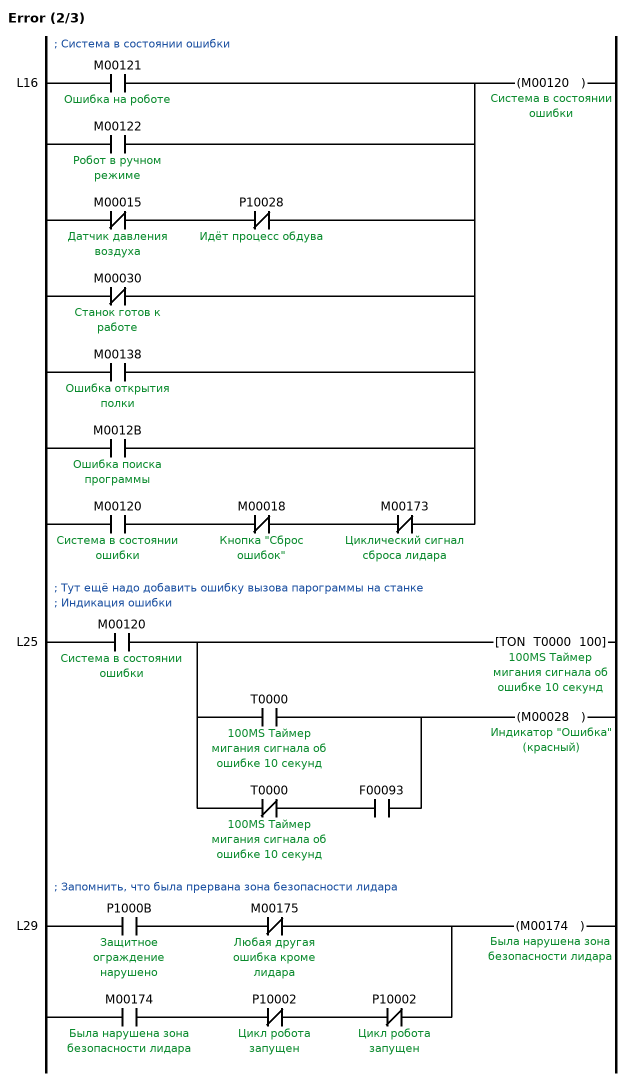
[picture p24: Error rungs L16-L29]
// Система в состоянии ошибки
; L16
LOAD      M00121	// Ошибка на роботе
OR        M00122	// Робот в ручном режиме
LOAD NOT  M00015	// Датчик давления воздуха
AND NOT   P10028	// Идёт процесс обдува
OR LOAD
OR NOT    M00030	// Станок готов к работе
OR        M00138	// Ошибка открытия полки
OR        M0012B	// Ошибка поиска программы
LOAD      M00120	// Система в состоянии ошибки
AND NOT   M00018	// Кнопка "Сброс ошибок"
AND NOT   M00173	// Циклический сигнал сброса лидара
OR LOAD
OUT       M00120	// Система в состоянии ошибки
// Тут ещё надо добавить ошибку вызова парограммы на станке
// Индикация ошибки
; L25
LOAD      M00120	// Система в состоянии ошибки
TON       T0000 100	// 100MS Таймер мигания сигнала об ошибке 10 секунд
LOAD      T0000	// 100MS Таймер мигания сигнала об ошибке 10 секунд
LOAD NOT  T0000	// 100MS Таймер мигания сигнала об ошибке 10 секунд
AND       F00093
OR LOAD
AND LOAD
OUT       M00028	// Индикатор "Ошибка" (красный)
// Запомнить, что была прервана зона безопасности лидара
; L29
LOAD      P1000B	// Защитное ограждение нарушено
AND NOT   M00175	// Любая другая ошибка кроме лидара
LOAD      M00174	// Была нарушена зона безопасности лидара
AND NOT   P10002	// Цикл робота запущен
AND NOT   P10002	// Цикл робота запущен
OR LOAD
OUT       M00174	// Была нарушена зона безопасности лидара

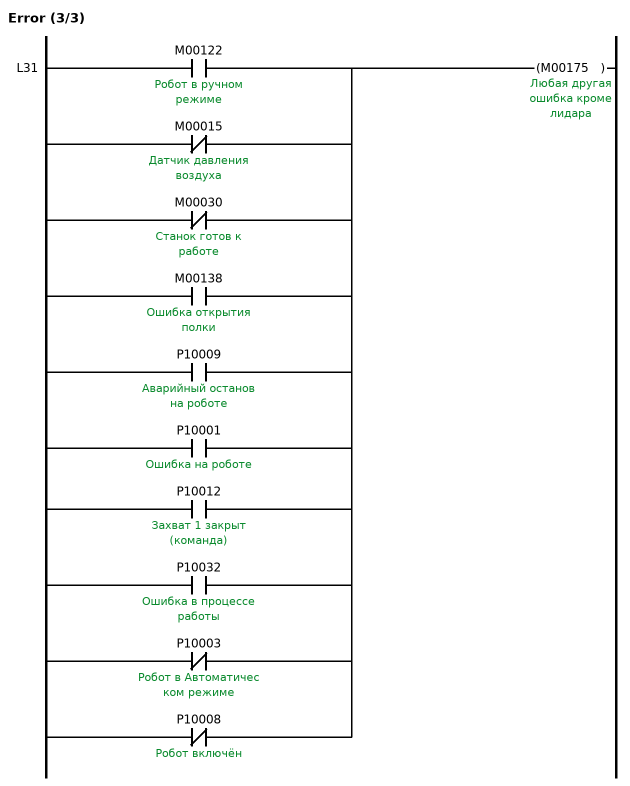
; L31
LOAD      M00122	// Робот в ручном режиме
OR NOT    M00015	// Датчик давления воздуха
OR NOT    M00030	// Станок готов к работе
OR        M00138	// Ошибка открытия полки
OR        P10009	// Аварийный останов на роботе
OR        P10001	// Ошибка на роботе
OR        P10012	// Захват 1 закрыт (команда)
OR        P10032	// Ошибка в процессе работы
OR NOT    P10003	// Робот в Автоматическом режиме
OR NOT    P10008	// Робот включён
OUT       M00175	// Любая другая ошибка кроме лидара

PROGRAM Shelves (task: Scan Program)

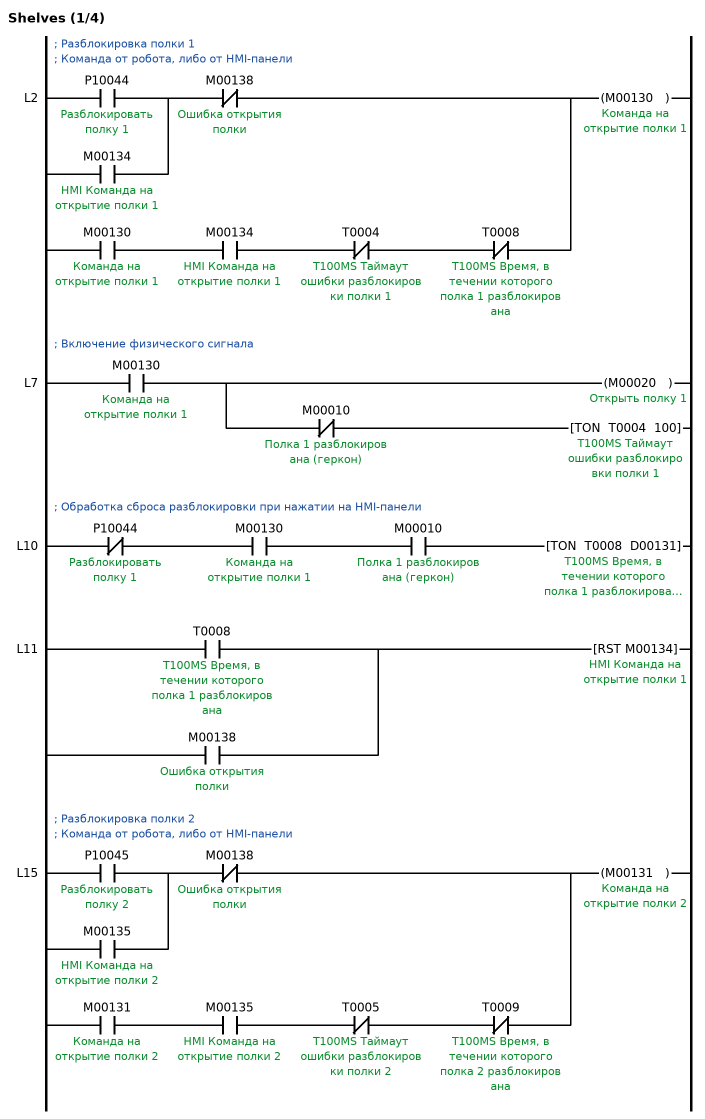
// Разблокировка полки 1
// Команда от робота, либо от HMI-панели
; L2
LOAD      P10044	// Разблокировать полку 1
OR        M00134	// HMI Команда на открытие полки 1
AND NOT   M00138	// Ошибка открытия полки
LOAD      M00130	// Команда на открытие полки 1
AND       M00134	// HMI Команда на открытие полки 1
AND NOT   T0004	// T100MS Таймаут ошибки разблокировки полки 1
AND NOT   T0008	// T100MS Время, в течении которого полка 1 разблокирована
OR LOAD
OUT       M00130	// Команда на открытие полки 1
// Включение физического сигнала
; L7
LOAD      M00130	// Команда на открытие полки 1
OUT       M00020	// Открыть полку 1
AND NOT   M00010	// Полка 1 разблокирована (геркон)
TON       T0004 100	// T100MS Таймаут ошибки разблокировки полки 1
// Обработка сброса разблокировки при нажатии на HMI-панели
; L10
LOAD NOT  P10044	// Разблокировать полку 1
AND       M00130	// Команда на открытие полки 1
AND       M00010	// Полка 1 разблокирована (геркон)
TON       T0008 D00131	// T100MS Время, в течении которого полка 1 разблокирована / HMI Время, в течении которого разблокирована полка после нажатия кнопки
; L11
LOAD      T0008	// T100MS Время, в течении которого полка 1 разблокирована
OR        M00138	// Ошибка открытия полки
RST       M00134	// HMI Команда на открытие полки 1
// Разблокировка полки 2
// Команда от робота, либо от HMI-панели
; L15
LOAD      P10045	// Разблокировать полку 2
OR        M00135	// HMI Команда на открытие полки 2
AND NOT   M00138	// Ошибка открытия полки
LOAD      M00131	// Команда на открытие полки 2
AND       M00135	// HMI Команда на открытие полки 2
AND NOT   T0005	// T100MS Таймаут ошибки разблокировки полки 2
AND NOT   T0009	// T100MS Время, в течении которого полка 2 разблокирована
OR LOAD
OUT       M00131	// Команда на открытие полки 2

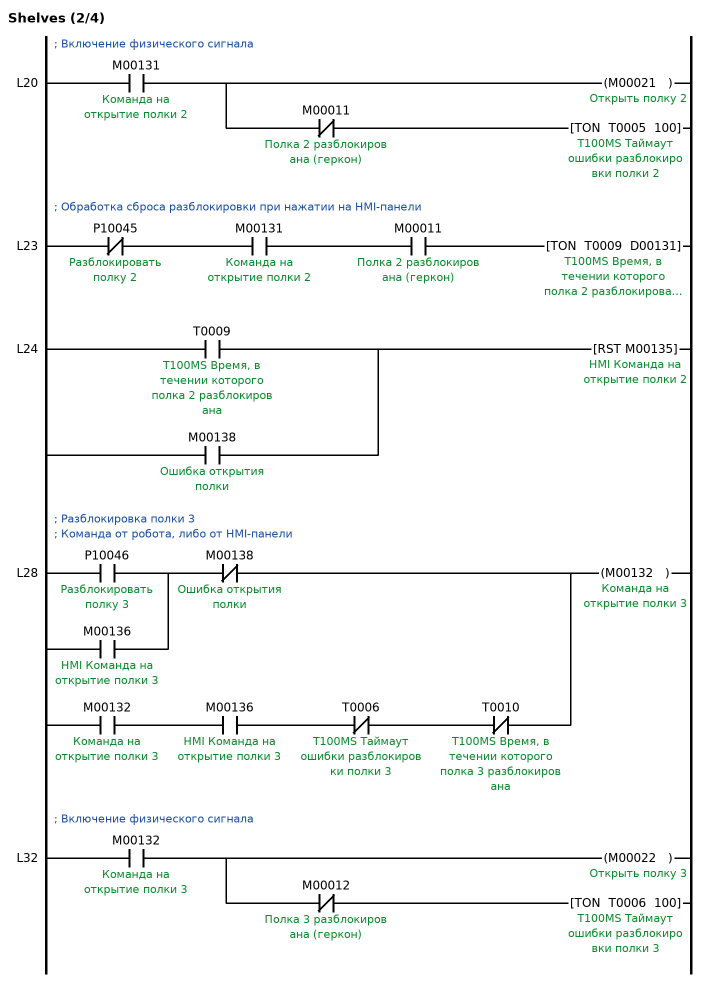
// Включение физического сигнала
; L20
LOAD      M00131	// Команда на открытие полки 2
OUT       M00021	// Открыть полку 2
AND NOT   M00011	// Полка 2 разблокирована (геркон)
TON       T0005 100	// T100MS Таймаут ошибки разблокировки полки 2
// Обработка сброса разблокировки при нажатии на HMI-панели
; L23
LOAD NOT  P10045	// Разблокировать полку 2
AND       M00131	// Команда на открытие полки 2
AND       M00011	// Полка 2 разблокирована (геркон)
TON       T0009 D00131	// T100MS Время, в течении которого полка 2 разблокирована / HMI Время, в течении которого разблокирована полка после нажатия кнопки
; L24
LOAD      T0009	// T100MS Время, в течении которого полка 2 разблокирована
OR        M00138	// Ошибка открытия полки
RST       M00135	// HMI Команда на открытие полки 2
// Разблокировка полки 3
// Команда от робота, либо от HMI-панели
; L28
LOAD      P10046	// Разблокировать полку 3
OR        M00136	// HMI Команда на открытие полки 3
AND NOT   M00138	// Ошибка открытия полки
LOAD      M00132	// Команда на открытие полки 3
AND       M00136	// HMI Команда на открытие полки 3
AND NOT   T0006	// T100MS Таймаут ошибки разблокировки полки 3
AND NOT   T0010	// T100MS Время, в течении которого полка 3 разблокирована
OR LOAD
OUT       M00132	// Команда на открытие полки 3
// Включение физического сигнала
; L32
LOAD      M00132	// Команда на открытие полки 3
OUT       M00022	// Открыть полку 3
AND NOT   M00012	// Полка 3 разблокирована (геркон)
TON       T0006 100	// T100MS Таймаут ошибки разблокировки полки 3

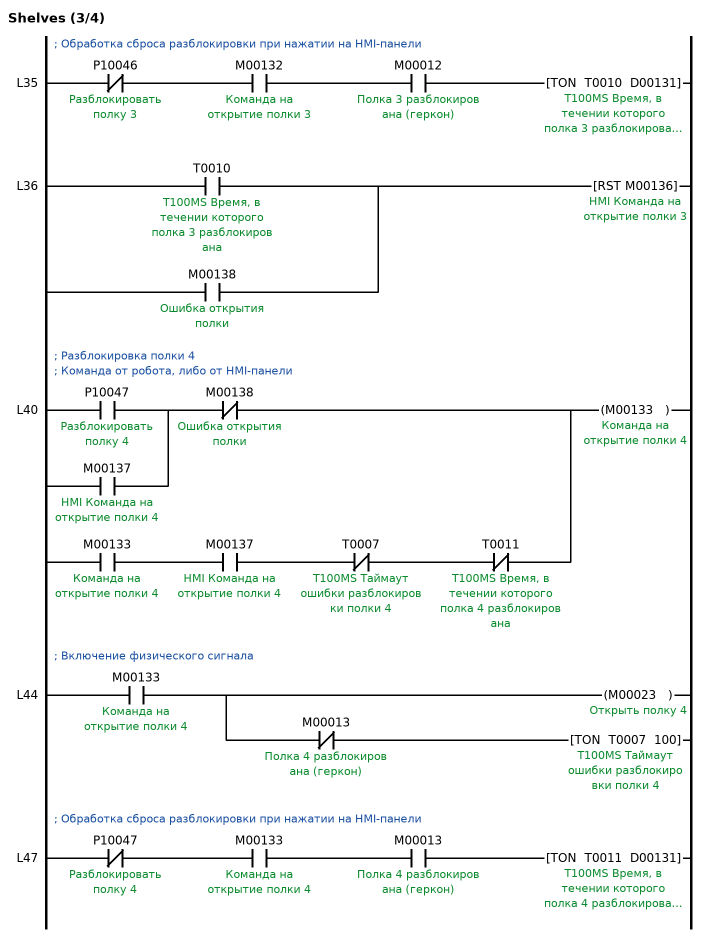
// Обработка сброса разблокировки при нажатии на HMI-панели
; L35
LOAD NOT  P10046	// Разблокировать полку 3
AND       M00132	// Команда на открытие полки 3
AND       M00012	// Полка 3 разблокирована (геркон)
TON       T0010 D00131	// T100MS Время, в течении которого полка 3 разблокирована / HMI Время, в течении которого разблокирована полка после нажатия кнопки
; L36
LOAD      T0010	// T100MS Время, в течении которого полка 3 разблокирована
OR        M00138	// Ошибка открытия полки
RST       M00136	// HMI Команда на открытие полки 3
// Разблокировка полки 4
// Команда от робота, либо от HMI-панели
; L40
LOAD      P10047	// Разблокировать полку 4
OR        M00137	// HMI Команда на открытие полки 4
AND NOT   M00138	// Ошибка открытия полки
LOAD      M00133	// Команда на открытие полки 4
AND       M00137	// HMI Команда на открытие полки 4
AND NOT   T0007	// T100MS Таймаут ошибки разблокировки полки 4
AND NOT   T0011	// T100MS Время, в течении которого полка 4 разблокирована
OR LOAD
OUT       M00133	// Команда на открытие полки 4
// Включение физического сигнала
; L44
LOAD      M00133	// Команда на открытие полки 4
OUT       M00023	// Открыть полку 4
AND NOT   M00013	// Полка 4 разблокирована (геркон)
TON       T0007 100	// T100MS Таймаут ошибки разблокировки полки 4
// Обработка сброса разблокировки при нажатии на HMI-панели
; L47
LOAD NOT  P10047	// Разблокировать полку 4
AND       M00133	// Команда на открытие полки 4
AND       M00013	// Полка 4 разблокирована (геркон)
TON       T0011 D00131	// T100MS Время, в течении которого полка 4 разблокирована / HMI Время, в течении которого разблокирована полка после нажатия кнопки

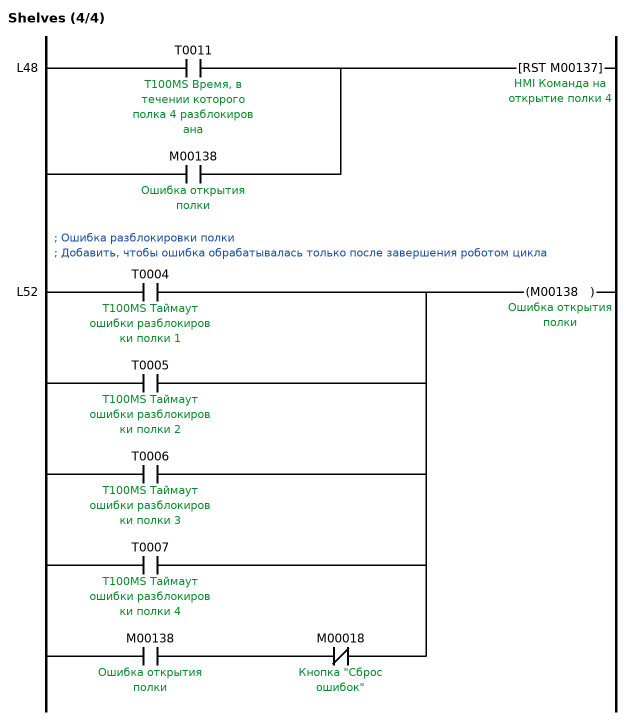
; L48
LOAD      T0011	// T100MS Время, в течении которого полка 4 разблокирована
OR        M00138	// Ошибка открытия полки
RST       M00137	// HMI Команда на открытие полки 4
// Ошибка разблокировки полки
// Добавить, чтобы ошибка обрабатывалась только после завершения роботом цикла
; L52
LOAD      T0004	// T100MS Таймаут ошибки разблокировки полки 1
OR        T0005	// T100MS Таймаут ошибки разблокировки полки 2
OR        T0006	// T100MS Таймаут ошибки разблокировки полки 3
OR        T0007	// T100MS Таймаут ошибки разблокировки полки 4
LOAD      M00138	// Ошибка открытия полки
AND NOT   M00018	// Кнопка "Сброс ошибок"
OR LOAD
OUT       M00138	// Ошибка открытия полки

PROGRAM Database (task: Scan Program)

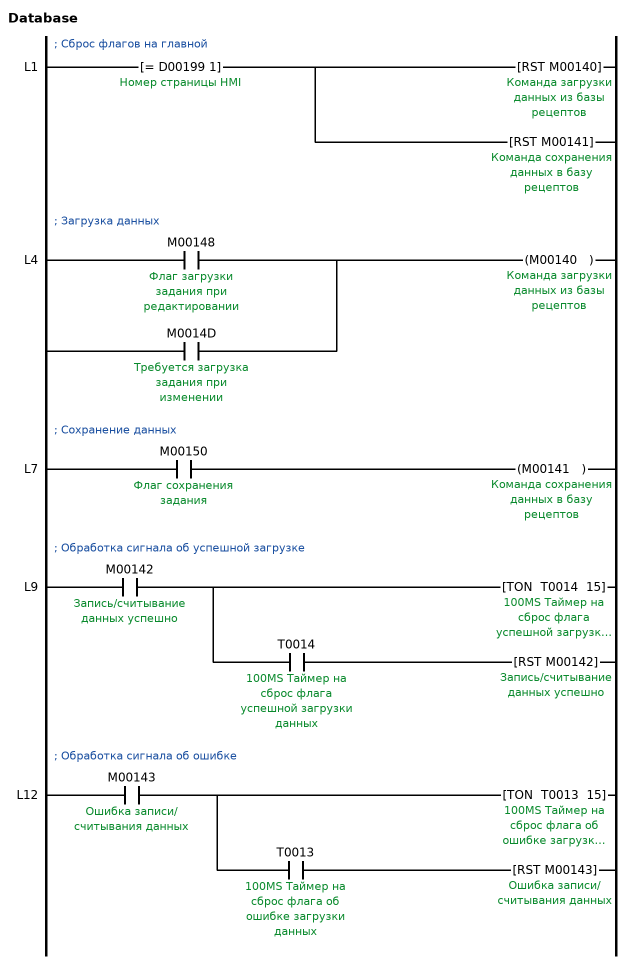
// Сброс флагов на главной
; L1
LOAD=     D00199 1	// Номер страницы HMI
RST       M00140	// Команда загрузки данных из базы рецептов
RST       M00141	// Команда сохранения данных в базу рецептов
// Загрузка данных
; L4
LOAD      M00148	// Флаг загрузки задания при редактировании
OR        M0014D	// Требуется загрузка задания при изменении
OUT       M00140	// Команда загрузки данных из базы рецептов
// Сохранение данных
; L7
LOAD      M00150	// Флаг сохранения задания
OUT       M00141	// Команда сохранения данных в базу рецептов
// Обработка сигнала об успешной загрузке
; L9
LOAD      M00142	// Запись/считывание данных успешно
TON       T0014 15	// 100MS Таймер на сброс флага успешной загрузки данных
AND       T0014	// 100MS Таймер на сброс флага успешной загрузки данных
RST       M00142	// Запись/считывание данных успешно
// Обработка сигнала об ошибке
; L12
LOAD      M00143	// Ошибка записи/считывания данных
TON       T0013 15	// 100MS Таймер на сброс флага об ошибке загрузки данных
AND       T0013	// 100MS Таймер на сброс флага об ошибке загрузки данных
RST       M00143	// Ошибка записи/считывания данных

PROGRAM HMI (task: Scan Program)

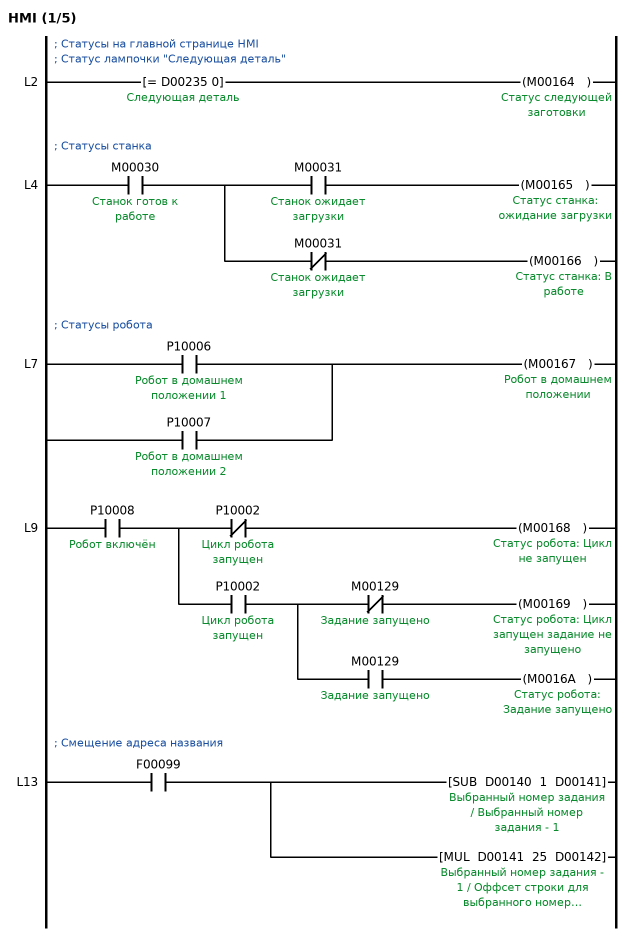
// Статусы на главной странице HMI
// Статус лампочки "Следующая деталь"
; L2
LOAD=     D00235 0	// Следующая деталь
OUT       M00164	// Статус следующей заготовки 
// Статусы станка
; L4
LOAD      M00030	// Станок готов к работе
MPUSH
AND       M00031	// Станок ожидает загрузки
OUT       M00165	// Статус станка: ожидание загрузки
MPOP
AND NOT   M00031	// Станок ожидает загрузки
OUT       M00166	// Статус станка: В работе
// Статусы робота
; L7
LOAD      P10006	// Робот в домашнем положении 1
OR        P10007	// Робот в домашнем положении 2
OUT       M00167	// Робот в домашнем положении
; L9
LOAD      P10008	// Робот включён
MPUSH
AND NOT   P10002	// Цикл робота запущен
OUT       M00168	// Статус робота: Цикл не запущен
MPOP
AND       P10002	// Цикл робота запущен
MPUSH
AND NOT   M00129	// Задание запущено
OUT       M00169	// Статус робота: Цикл запущен задание не запущено
MPOP
AND       M00129	// Задание запущено
OUT       M0016A	// Статус робота: Задание запущено
// Смещение адреса названия
; L13
LOAD      F00099
SUB       D00140 1 D00141	// Выбранный номер задания / Выбранный номер задания - 1
MUL       D00141 25 D00142	// Выбранный номер задания - 1 / Оффсет строки для выбранного номера названия

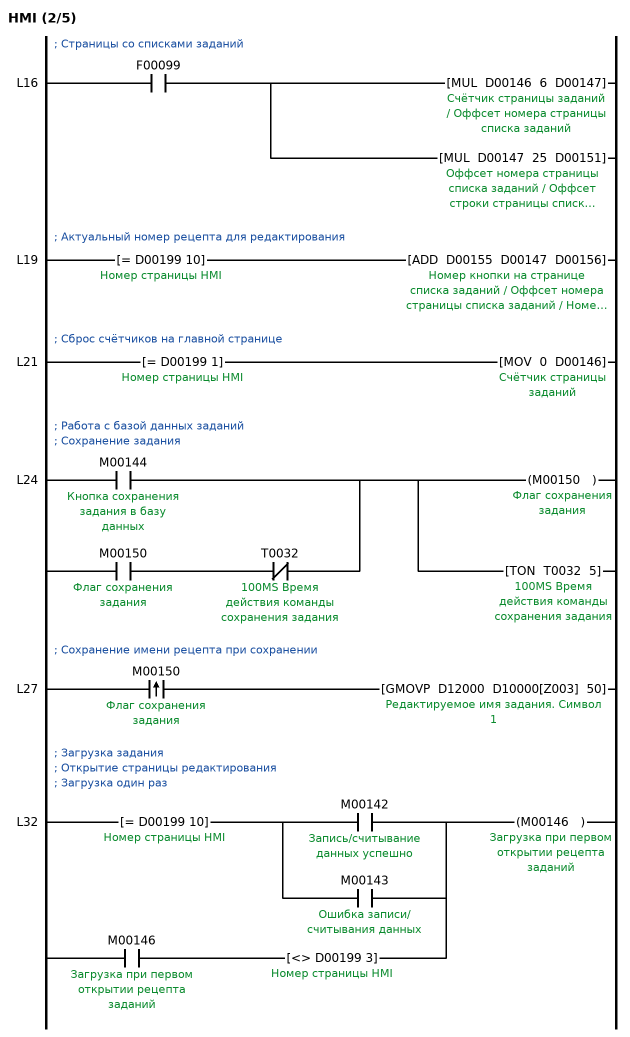
// Страницы со списками заданий
; L16
LOAD      F00099
MUL       D00146 6 D00147	// Счётчик страницы заданий / Оффсет номера страницы списка заданий
MUL       D00147 25 D00151	// Оффсет номера страницы списка заданий / Оффсет строки страницы списка заданий
// Актуальный номер рецепта для редактирования
; L19
LOAD=     D00199 10	// Номер страницы HMI
ADD       D00155 D00147 D00156	// Номер кнопки на странице списка заданий / Оффсет номера страницы списка заданий / Номер редактируемого задания
// Сброс счётчиков на главной странице
; L21
LOAD=     D00199 1	// Номер страницы HMI
MOV       0 D00146	// Счётчик страницы заданий
// Работа с базой данных заданий
// Сохранение задания
; L24
LOAD      M00144	// Кнопка сохранения задания в базу данных
LOAD      M00150	// Флаг сохранения задания
AND NOT   T0032	// 100MS Время действия команды сохранения задания
OR LOAD
OUT       M00150	// Флаг сохранения задания
TON       T0032 5	// 100MS Время действия команды сохранения задания
// Сохранение имени рецепта при сохранении
; L27
LOADP     M00150	// Флаг сохранения задания
GMOVP     D12000 D10000[Z003] 50	// Редактируемое имя задания. Символ 1
// Загрузка задания
// Открытие страницы редактирования
// Загрузка один раз
; L32
LOAD=     D00199 10	// Номер страницы HMI
LOAD      M00142	// Запись/считывание данных успешно
OR        M00143	// Ошибка записи/считывания данных
AND LOAD
LOAD      M00146	// Загрузка при первом открытии рецепта заданий
AND<>     D00199 3	// Номер страницы HMI
OR LOAD
OUT       M00146	// Загрузка при первом открытии рецепта заданий

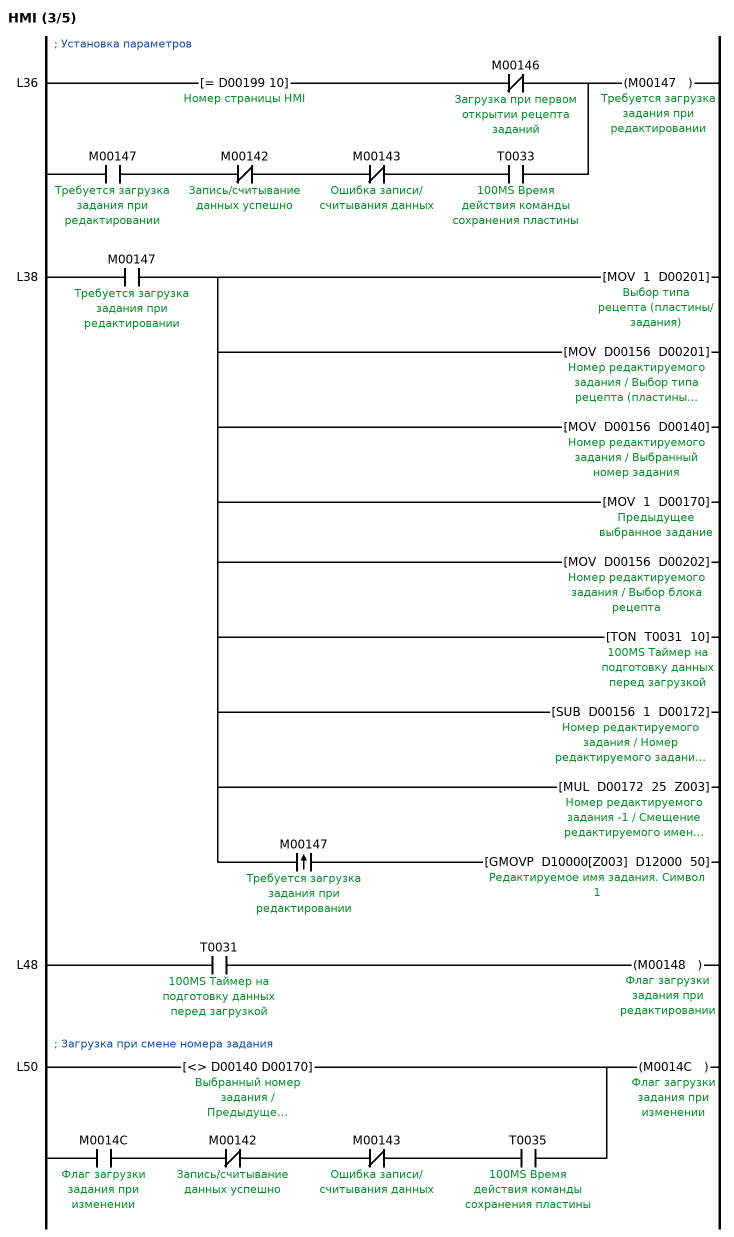
// Установка параметров
; L36
LOAD=     D00199 10	// Номер страницы HMI
AND NOT   M00146	// Загрузка при первом открытии рецепта заданий
LOAD      M00147	// Требуется загрузка задания при редактировании
AND NOT   M00142	// Запись/считывание данных успешно
AND NOT   M00143	// Ошибка записи/считывания данных
AND       T0033	// 100MS Время действия команды сохранения пластины
OR LOAD
OUT       M00147	// Требуется загрузка задания при редактировании
; L38
LOAD      M00147	// Требуется загрузка задания при редактировании
MOV       1 D00201	// Выбор типа рецепта (пластины/задания)
MOV       D00156 D00201	// Номер редактируемого задания / Выбор типа рецепта (пластины/задания)
MOV       D00156 D00140	// Номер редактируемого задания / Выбранный номер задания
MOV       1 D00170	// Предыдущее выбранное задание
MOV       D00156 D00202	// Номер редактируемого задания / Выбор блока рецепта
TON       T0031 10	// 100MS Таймер на подготовку данных перед загрузкой
SUB       D00156 1 D00172	// Номер редактируемого задания / Номер редактируемого задания -1
MUL       D00172 25 Z003	// Номер редактируемого задания -1 / Смещение редактируемого имени задания
ANDP      M00147	// Требуется загрузка задания при редактировании
GMOVP     D10000[Z003] D12000 50	// Редактируемое имя задания. Символ 1
; L48
LOAD      T0031	// 100MS Таймер на подготовку данных перед загрузкой
OUT       M00148	// Флаг загрузки задания при редактировании
// Загрузка при смене номера задания
; L50
LOAD<>    D00140 D00170	// Выбранный номер задания / Предыдущее выбранное задание
LOAD      M0014C	// Флаг загрузки задания при изменении
AND NOT   M00142	// Запись/считывание данных успешно
AND NOT   M00143	// Ошибка записи/считывания данных
AND       T0035	// 100MS Время действия команды сохранения пластины
OR LOAD
OUT       M0014C	// Флаг загрузки задания при изменении

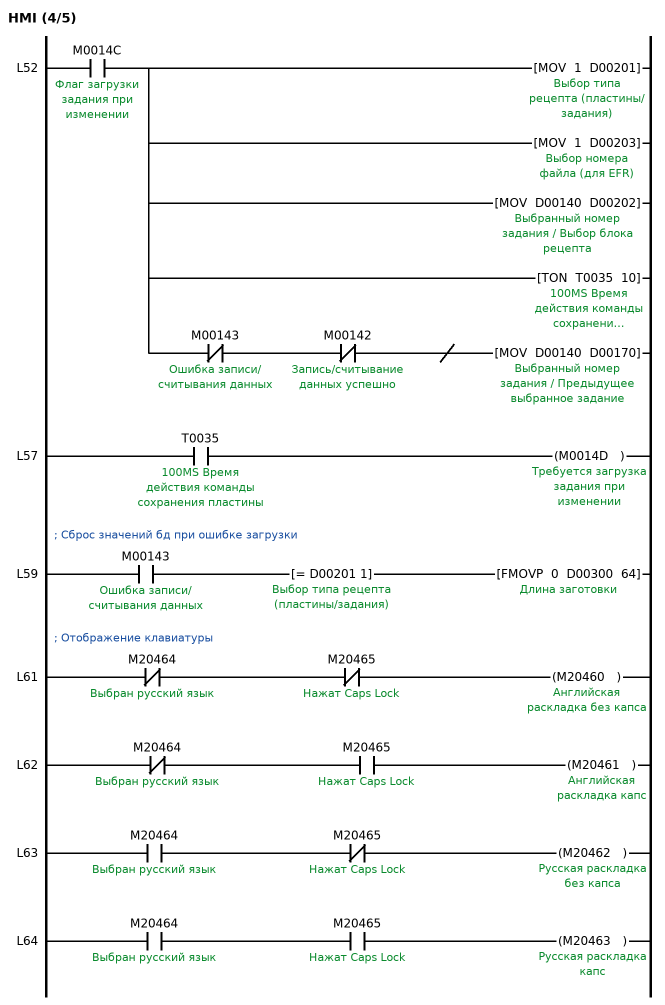
; L52
LOAD      M0014C	// Флаг загрузки задания при изменении
MOV       1 D00201	// Выбор типа рецепта (пластины/задания)
MOV       1 D00203	// Выбор номера файла (для EFR)
MOV       D00140 D00202	// Выбранный номер задания / Выбор блока рецепта
TON       T0035 10	// 100MS Время действия команды сохранения пластины
AND NOT   M00143	// Ошибка записи/считывания данных
AND NOT   M00142	// Запись/считывание данных успешно
NOT
MOV       D00140 D00170	// Выбранный номер задания / Предыдущее выбранное задание
; L57
LOAD      T0035	// 100MS Время действия команды сохранения пластины
OUT       M0014D	// Требуется загрузка задания при изменении
// Сброс значений бд при ошибке загрузки
; L59
LOAD      M00143	// Ошибка записи/считывания данных
AND=      D00201 1	// Выбор типа рецепта (пластины/задания)
FMOVP     0 D00300 64	// Длина заготовки
// Отображение клавиатуры
; L61
LOAD NOT  M20464	// Выбран русский язык
AND NOT   M20465	// Нажат Caps Lock
OUT       M20460	// Английская раскладка без капса
; L62
LOAD NOT  M20464	// Выбран русский язык
AND       M20465	// Нажат Caps Lock
OUT       M20461	// Английская раскладка капс
; L63
LOAD      M20464	// Выбран русский язык
AND NOT   M20465	// Нажат Caps Lock
OUT       M20462	// Русская раскладка без капса
; L64
LOAD      M20464	// Выбран русский язык
AND       M20465	// Нажат Caps Lock
OUT       M20463	// Русская раскладка капс

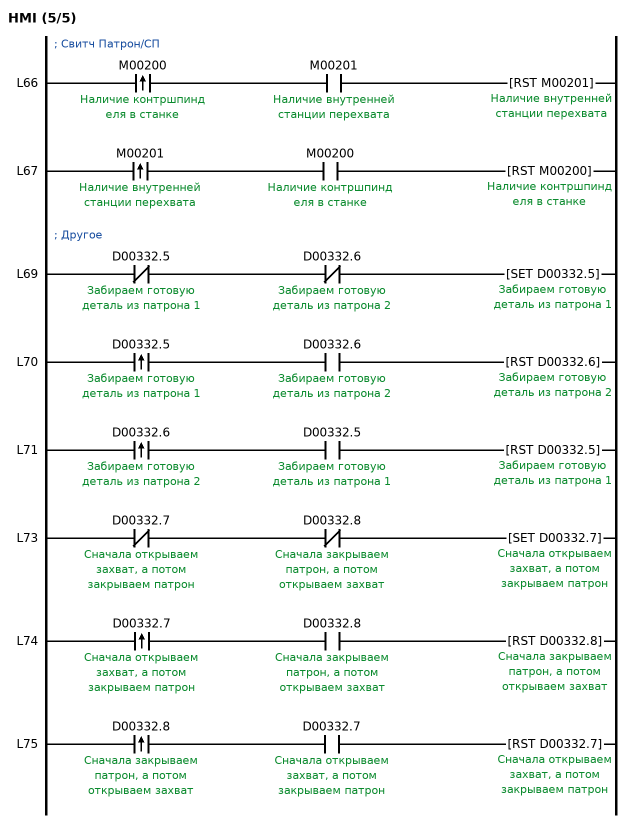
// Свитч Патрон/СП
; L66
LOADP     M00200	// Наличие контршпинделя в станке
AND       M00201	// Наличие внутренней станции перехвата
RST       M00201	// Наличие внутренней станции перехвата
; L67
LOADP     M00201	// Наличие внутренней станции перехвата
AND       M00200	// Наличие контршпинделя в станке
RST       M00200	// Наличие контршпинделя в станке
// Другое
; L69
LOAD NOT  D00332.5	// Забираем готовую деталь из патрона 1
AND NOT   D00332.6	// Забираем готовую деталь из патрона 2
SET       D00332.5	// Забираем готовую деталь из патрона 1
; L70
LOADP     D00332.5	// Забираем готовую деталь из патрона 1
AND       D00332.6	// Забираем готовую деталь из патрона 2
RST       D00332.6	// Забираем готовую деталь из патрона 2
; L71
LOADP     D00332.6	// Забираем готовую деталь из патрона 2
AND       D00332.5	// Забираем готовую деталь из патрона 1
RST       D00332.5	// Забираем готовую деталь из патрона 1
; L73
LOAD NOT  D00332.7	// Сначала открываем захват, а потом закрываем патрон
AND NOT   D00332.8	// Сначала закрываем патрон, а потом открываем захват
SET       D00332.7	// Сначала открываем захват, а потом закрываем патрон
; L74
LOADP     D00332.7	// Сначала открываем захват, а потом закрываем патрон
AND       D00332.8	// Сначала закрываем патрон, а потом открываем захват
RST       D00332.8	// Сначала закрываем патрон, а потом открываем захват
; L75
LOADP     D00332.8	// Сначала закрываем патрон, а потом открываем захват
AND       D00332.7	// Сначала открываем захват, а потом закрываем патрон
RST       D00332.7	// Сначала открываем захват, а потом закрываем патрон

PROGRAM Initialization (task: Scan Program)

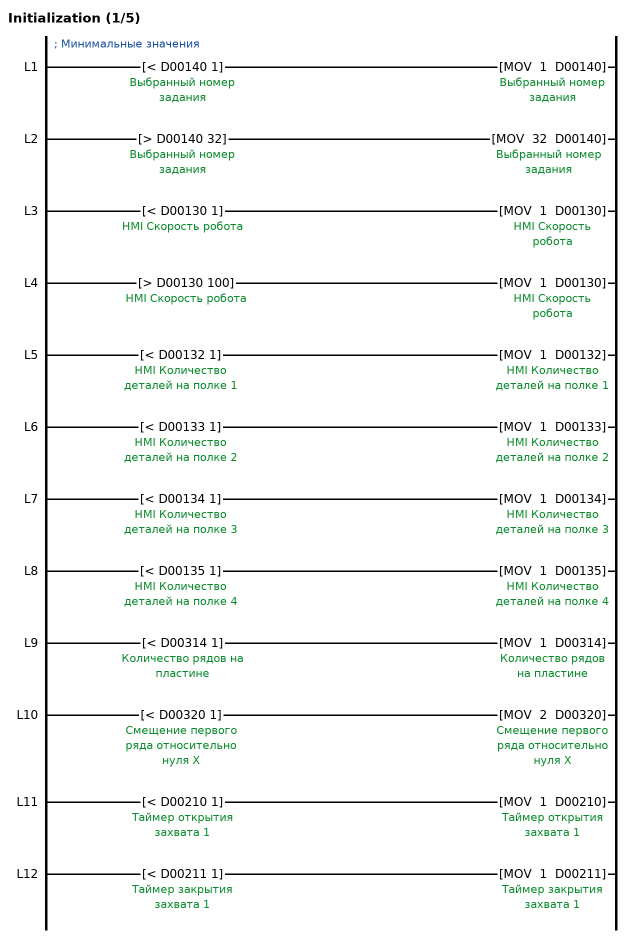
// Минимальные значения
; L1
LOAD<     D00140 1	// Выбранный номер задания
MOV       1 D00140	// Выбранный номер задания
; L2
LOAD>     D00140 32	// Выбранный номер задания
MOV       32 D00140	// Выбранный номер задания
; L3
LOAD<     D00130 1	// HMI Скорость робота
MOV       1 D00130	// HMI Скорость робота
; L4
LOAD>     D00130 100	// HMI Скорость робота
MOV       1 D00130	// HMI Скорость робота
; L5
LOAD<     D00132 1	// HMI Количество деталей на полке 1
MOV       1 D00132	// HMI Количество деталей на полке 1
; L6
LOAD<     D00133 1	// HMI Количество деталей на полке 2
MOV       1 D00133	// HMI Количество деталей на полке 2
; L7
LOAD<     D00134 1	// HMI Количество деталей на полке 3
MOV       1 D00134	// HMI Количество деталей на полке 3
; L8
LOAD<     D00135 1	// HMI Количество деталей на полке 4
MOV       1 D00135	// HMI Количество деталей на полке 4
; L9
LOAD<     D00314 1	// Количество рядов на пластине
MOV       1 D00314	// Количество рядов на пластине
; L10
LOAD<     D00320 1	// Смещение первого ряда относительно нуля Х
MOV       2 D00320	// Смещение первого ряда относительно нуля Х
; L11
LOAD<     D00210 1	// Таймер открытия захвата 1
MOV       1 D00210	// Таймер открытия захвата 1
; L12
LOAD<     D00211 1	// Таймер закрытия захвата 1
MOV       1 D00211	// Таймер закрытия захвата 1

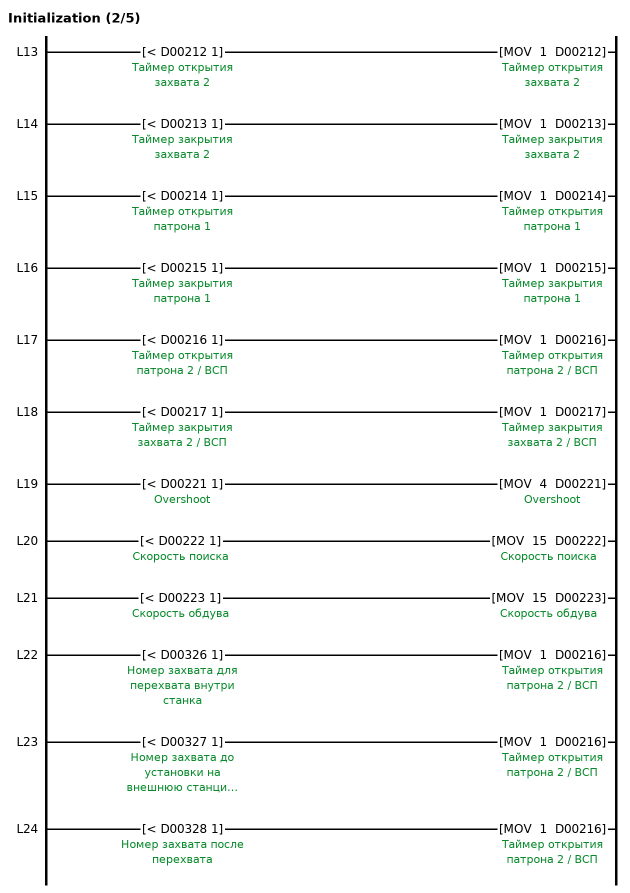
; L13
LOAD<     D00212 1	// Таймер открытия захвата 2
MOV       1 D00212	// Таймер открытия захвата 2
; L14
LOAD<     D00213 1	// Таймер закрытия захвата 2
MOV       1 D00213	// Таймер закрытия захвата 2
; L15
LOAD<     D00214 1	// Таймер открытия патрона 1
MOV       1 D00214	// Таймер открытия патрона 1
; L16
LOAD<     D00215 1	// Таймер закрытия патрона 1
MOV       1 D00215	// Таймер закрытия патрона 1
; L17
LOAD<     D00216 1	// Таймер открытия патрона 2 / ВСП
MOV       1 D00216	// Таймер открытия патрона 2 / ВСП
; L18
LOAD<     D00217 1	// Таймер закрытия захвата 2 / ВСП
MOV       1 D00217	// Таймер закрытия захвата 2 / ВСП
; L19
LOAD<     D00221 1	// Overshoot
MOV       4 D00221	// Overshoot
; L20
LOAD<     D00222 1	// Скорость поиска
MOV       15 D00222	// Скорость поиска
; L21
LOAD<     D00223 1	// Скорость обдува
MOV       15 D00223	// Скорость обдува
; L22
LOAD<     D00326 1	// Номер захвата для перехвата внутри станка
MOV       1 D00216	// Таймер открытия патрона 2 / ВСП
; L23
LOAD<     D00327 1	// Номер захвата до установки на внешнюю станцию перехвата
MOV       1 D00216	// Таймер открытия патрона 2 / ВСП
; L24
LOAD<     D00328 1	// Номер захвата после перехвата
MOV       1 D00216	// Таймер открытия патрона 2 / ВСП

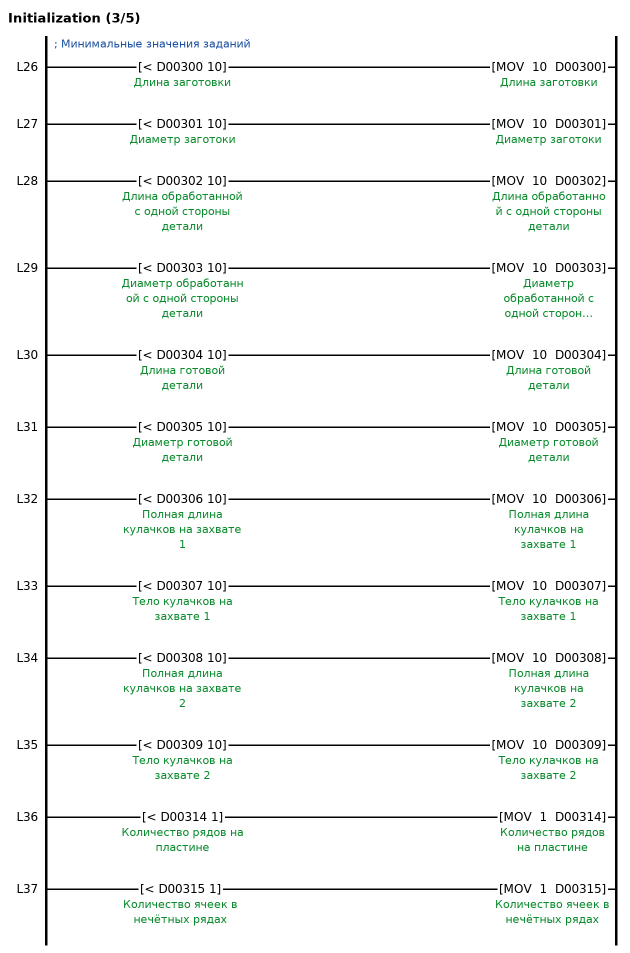
// Минимальные значения заданий
; L26
LOAD<     D00300 10	// Длина заготовки
MOV       10 D00300	// Длина заготовки
; L27
LOAD<     D00301 10	// Диаметр заготоки
MOV       10 D00301	// Диаметр заготоки
; L28
LOAD<     D00302 10	// Длина обработанной с одной стороны детали
MOV       10 D00302	// Длина обработанной с одной стороны детали
; L29
LOAD<     D00303 10	// Диаметр обработанной с одной стороны детали
MOV       10 D00303	// Диаметр обработанной с одной стороны детали
; L30
LOAD<     D00304 10	// Длина готовой детали
MOV       10 D00304	// Длина готовой детали
; L31
LOAD<     D00305 10	// Диаметр готовой детали
MOV       10 D00305	// Диаметр готовой детали
; L32
LOAD<     D00306 10	// Полная длина кулачков на захвате 1
MOV       10 D00306	// Полная длина кулачков на захвате 1
; L33
LOAD<     D00307 10	// Тело кулачков на захвате 1
MOV       10 D00307	// Тело кулачков на захвате 1
; L34
LOAD<     D00308 10	// Полная длина кулачков на захвате 2
MOV       10 D00308	// Полная длина кулачков на захвате 2
; L35
LOAD<     D00309 10	// Тело кулачков на захвате 2
MOV       10 D00309	// Тело кулачков на захвате 2
; L36
LOAD<     D00314 1	// Количество рядов на пластине
MOV       1 D00314	// Количество рядов на пластине
; L37
LOAD<     D00315 1	// Количество ячеек в нечётных рядах
MOV       1 D00315	// Количество ячеек в нечётных рядах

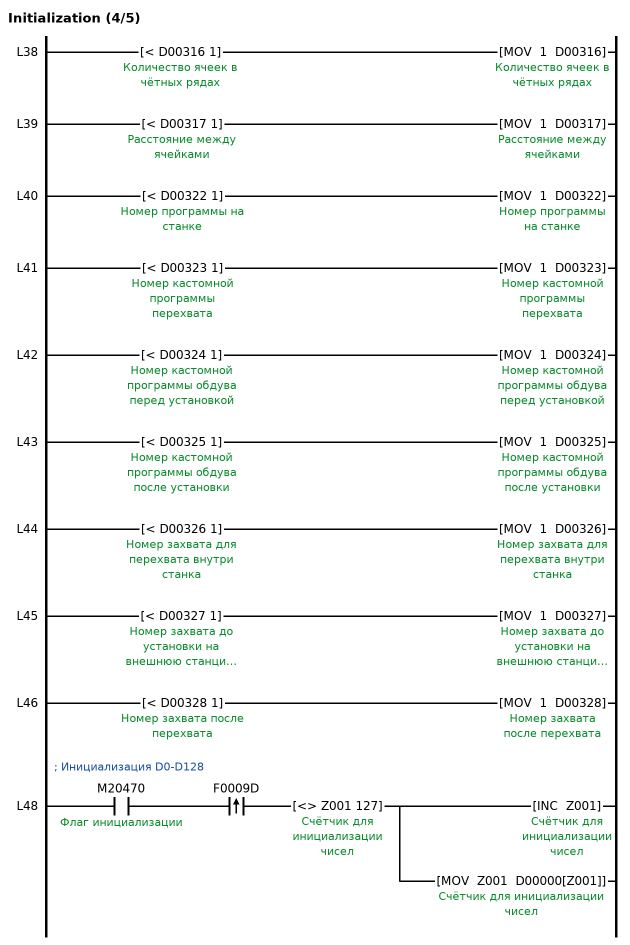
; L38
LOAD<     D00316 1	// Количество ячеек в чётных рядах
MOV       1 D00316	// Количество ячеек в чётных рядах
; L39
LOAD<     D00317 1	// Расстояние между ячейками
MOV       1 D00317	// Расстояние между ячейками
; L40
LOAD<     D00322 1	// Номер программы на станке
MOV       1 D00322	// Номер программы на станке
; L41
LOAD<     D00323 1	// Номер кастомной программы перехвата
MOV       1 D00323	// Номер кастомной программы перехвата
; L42
LOAD<     D00324 1	// Номер кастомной программы обдува перед установкой
MOV       1 D00324	// Номер кастомной программы обдува перед установкой
; L43
LOAD<     D00325 1	// Номер кастомной программы обдува после установки
MOV       1 D00325	// Номер кастомной программы обдува после установки
; L44
LOAD<     D00326 1	// Номер захвата для перехвата внутри станка
MOV       1 D00326	// Номер захвата для перехвата внутри станка
; L45
LOAD<     D00327 1	// Номер захвата до установки на внешнюю станцию перехвата
MOV       1 D00327	// Номер захвата до установки на внешнюю станцию перехвата
; L46
LOAD<     D00328 1	// Номер захвата после перехвата
MOV       1 D00328	// Номер захвата после перехвата
// Инициализация D0-D128
; L48
LOAD      M20470	// Флаг инициализации
ANDP      F0009D
AND<>     Z001 127	// Счётчик для инициализации чисел
INC       Z001	// Счётчик для инициализации чисел
MOV       Z001 D00000[Z001]	// Счётчик для инициализации чисел

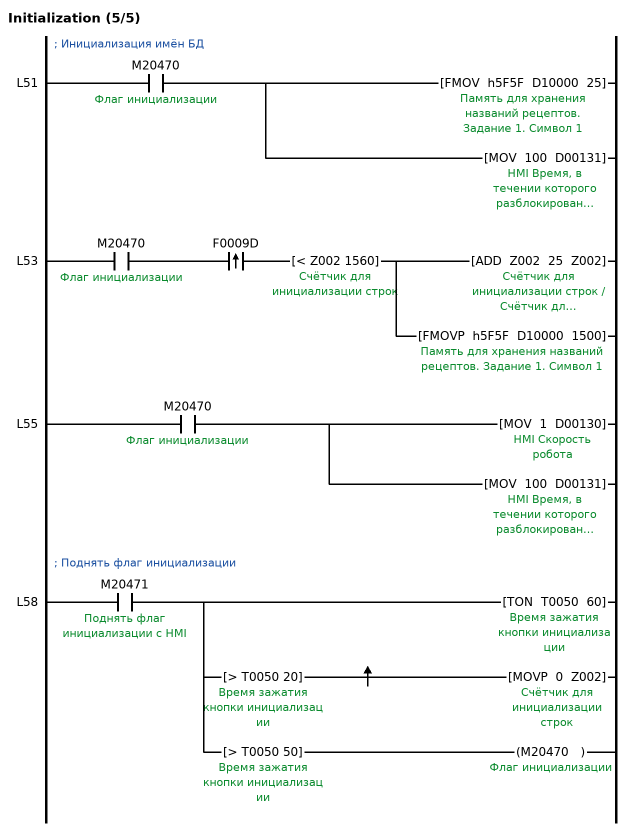
// Инициализация имён БД
; L51
LOAD      M20470	// Флаг инициализации
FMOV      h5F5F D10000 25	// Память для хранения названий рецептов. Задание 1. Символ 1
MOV       100 D00131	// HMI Время, в течении которого разблокирована полка после нажатия кнопки
; L53
LOAD      M20470	// Флаг инициализации
ANDP      F0009D
AND<      Z002 1560	// Счётчик для инициализации строк
ADD       Z002 25 Z002	// Счётчик для инициализации строк / Счётчик для инициализации строк
FMOVP     h5F5F D10000 1500	// Память для хранения названий рецептов. Задание 1. Символ 1
; L55
LOAD      M20470	// Флаг инициализации
MOV       1 D00130	// HMI Скорость робота
MOV       100 D00131	// HMI Время, в течении которого разблокирована полка после нажатия кнопки
// Поднять флаг инициализации
; L58
LOAD      M20471	// Поднять флаг инициализации с HMI
TON       T0050 60	// Время зажатия кнопки инициализации
MPUSH
AND>      T0050 20	// Время зажатия кнопки инициализации
R_EDGE
MOVP      0 Z002	// Счётчик для инициализации строк
MPOP
AND>      T0050 50	// Время зажатия кнопки инициализации
OUT       M20470	// Флаг инициализации

VARIABLES AND COMMENTS (devices not used above)
P1000C	BIT	Требуется замена батареи питания энкодера
D00000	WORD	Фиксированное число 0
D00001	WORD	Фиксированное число 1
D00002	WORD	Фиксированное число 2
D00003	WORD	Фиксированное число 3
D00004	WORD	Фиксированное число 4
D00005	WORD	Фиксированное число 5
D00006	WORD	Фиксированное число 6
D00007	WORD	Фиксированное число 7
D00008	WORD	Фиксированное число 8
D00009	WORD	Фиксированное число 9
D00010	WORD	Фиксированное число 10
D00011	WORD	Фиксированное число 11
D00012	WORD	Фиксированное число 12
D00013	WORD	Фиксированное число 13
D00014	WORD	Фиксированное число 14
D00015	WORD	Фиксированное число 15
D00016	WORD	Фиксированное число 16
D00017	WORD	Фиксированное число 17
D00018	WORD	Фиксированное число 18
D00019	WORD	Фиксированное число 19
D00020	WORD	Фиксированное число 20
D00021	WORD	Фиксированное число 21
D00022	WORD	Фиксированное число 22
D00023	WORD	Фиксированное число 23
D00024	WORD	Фиксированное число 24
D00025	WORD	Фиксированное число 25
D00026	WORD	Фиксированное число 26
D00027	WORD	Фиксированное число 27
D00028	WORD	Фиксированное число 28
D00029	WORD	Фиксированное число 29
D00030	WORD	Фиксированное число 30
D00031	WORD	Фиксированное число 31
D00032	WORD	Фиксированное число 32
D00033	WORD	Фиксированное число 33
D00034	WORD	Фиксированное число 34
D00035	WORD	Фиксированное число 35
D00036	WORD	Фиксированное число 36
D00037	WORD	Фиксированное число 37
D00038	WORD	Фиксированное число 38
D00039	WORD	Фиксированное число 39
D00040	WORD	Фиксированное число 40
D00041	WORD	Фиксированное число 41
D00042	WORD	Фиксированное число 42
D00043	WORD	Фиксированное число 43
D00044	WORD	Фиксированное число 44
D00045	WORD	Фиксированное число 45
D00046	WORD	Фиксированное число 46
D00047	WORD	Фиксированное число 47
D00048	WORD	Фиксированное число 48
D00049	WORD	Фиксированное число 49
D00050	WORD	Фиксированное число 50
D00051	WORD	Фиксированное число 51
D00052	WORD	Фиксированное число 52
D00053	WORD	Фиксированное число 53
D00054	WORD	Фиксированное число 54
D00055	WORD	Фиксированное число 55
D00056	WORD	Фиксированное число 56
D00057	WORD	Фиксированное число 57
D00058	WORD	Фиксированное число 58
D00059	WORD	Фиксированное число 59
D00060	WORD	Фиксированное число 60
D00061	WORD	Фиксированное число 61
D00062	WORD	Фиксированное число 62
D00063	WORD	Фиксированное число 63
D00064	WORD	Фиксированное число 64
D00065	WORD	Фиксированное число 65
D00066	WORD	Фиксированное число 66
D00067	WORD	Фиксированное число 67
D00068	WORD	Фиксированное число 68
D00069	WORD	Фиксированное число 69
D00070	WORD	Фиксированное число 70
D00071	WORD	Фиксированное число 71
D00072	WORD	Фиксированное число 72
D00073	WORD	Фиксированное число 73
D00074	WORD	Фиксированное число 74
D00075	WORD	Фиксированное число 75
D00076	WORD	Фиксированное число 76
D00077	WORD	Фиксированное число 77
D00078	WORD	Фиксированное число 78
D00079	WORD	Фиксированное число 79
D00080	WORD	Фиксированное число 80
D00081	WORD	Фиксированное число 81
D00082	WORD	Фиксированное число 82
D00083	WORD	Фиксированное число 83
D00084	WORD	Фиксированное число 84
D00085	WORD	Фиксированное число 85
D00086	WORD	Фиксированное число 86
D00087	WORD	Фиксированное число 87
D00088	WORD	Фиксированное число 88
D00089	WORD	Фиксированное число 89
D00090	WORD	Фиксированное число 90
D00091	WORD	Фиксированное число 91
D00092	WORD	Фиксированное число 92
D00093	WORD	Фиксированное число 93
D00094	WORD	Фиксированное число 94
D00095	WORD	Фиксированное число 95
D00096	WORD	Фиксированное число 96
D00097	WORD	Фиксированное число 97
D00098	WORD	Фиксированное число 98
D00099	WORD	Фиксированное число 99
D00100	WORD	Фиксированное число 100
D00101	WORD	Фиксированное число 101
D00102	WORD	Фиксированное число 102
D00103	WORD	Фиксированное число 103
D00104	WORD	Фиксированное число 104
D00105	WORD	Фиксированное число 105
D00106	WORD	Фиксированное число 106
D00107	WORD	Фиксированное число 107
D00108	WORD	Фиксированное число 108
D00109	WORD	Фиксированное число 109
D00110	WORD	Фиксированное число 110
D00111	WORD	Фиксированное число 111
D00112	WORD	Фиксированное число 112
D00113	WORD	Фиксированное число 113
D00114	WORD	Фиксированное число 114
D00115	WORD	Фиксированное число 115
D00116	WORD	Фиксированное число 116
D00117	WORD	Фиксированное число 117
D00118	WORD	Фиксированное число 118
D00119	WORD	Фиксированное число 119
D00120	WORD	Фиксированное число 120
D00121	WORD	Фиксированное число 121
D00122	WORD	Фиксированное число 122
D00123	WORD	Фиксированное число 123
D00124	WORD	Фиксированное число 124
D00125	WORD	Фиксированное число 125
D00126	WORD	Фиксированное число 126
D00127	WORD	Фиксированное число 127
D00128	WORD	Фиксированное число 128
P1110	WORD	Таймер открытия патрона 1 (0)
P10010	BIT	Захват 1 открыт (датчик)
P10011	BIT	Захват 1 открыт (команда)
P10013	BIT	Ошибка открытия захвата 1 (при наличии датчика)
P10014	BIT	Усилие на захвате 1 (датчик)
P10030	BIT	Робот готов к запуску задания
P11010	BIT	Открыть захват 1 с HMI
P11011	BIT	Закрыть захват 1 с HMI
M00139	BIT	Индикатор ошибки открытия полки
P10037	BIT	Данные с ПЛК считаны
P10040	BIT	Полка 1 открыта
P10041	BIT	Полка 2 открыта
P10042	BIT	Полка 3 открыта
P10043	BIT	Полка 4 открыта
P11100	BIT	Таймер открытия патрона 1 (0)
D00200	WORD	Код ошибки работы с базой данных
D00329	WORD	Резерв
D00330	WORD	Резерв
M00160	BIT	Статус захвата 1
M00161	BIT	Статус захвата 2
M00162	BIT	Статус патрона 1
M00163	BIT	Статус патрона 2
D00143	WORD	MULNULL
D00144	WORD	MULNULL
D00145	WORD	MULNULL
D00148	WORD	MULNULL
D00149	WORD	MULNULL
D00150	WORD	MULNULL
D00152	WORD	MULNULL
D00153	WORD	MULNULL
D00154	WORD	MULNULL
D00157	WORD	Счётчик страницы пластин
D00158	WORD	Оффсет номера страницы списка пластин
D00159	WORD	MULNULL
D00160	WORD	MULNULL
D00161	WORD	MULNULL
D00162	WORD	Оффсет строки страницы списка пластин
D00163	WORD	MULNULL
D00164	WORD	MULNULL
D00165	WORD	MULNULL
D00166	WORD	Номер кнопки на странице списка пластин
D00167	WORD	Номер редактируемой пластины
D10001	WORD	Память для хранения названий рецептов. Задание 1. Символ 2
D10002	WORD	Память для хранения названий рецептов. Задание 1. Символ 3
D10003	WORD	Память для хранения названий рецептов. Задание 1. Символ 4
D10004	WORD	Память для хранения названий рецептов. Задание 1. Символ 5
D10005	WORD	Память для хранения названий рецептов. Задание 1. Символ 6
D10006	WORD	Память для хранения названий рецептов. Задание 1. Символ 7
D10007	WORD	Память для хранения названий рецептов. Задание 1. Символ 8
D10008	WORD	Память для хранения названий рецептов. Задание 1. Символ 9
D10009	WORD	Память для хранения названий рецептов. Задание 1. Символ 10
D10010	WORD	Память для хранения названий рецептов. Задание 1. Символ 11
D10011	WORD	Память для хранения названий рецептов. Задание 1. Символ 12
D10012	WORD	Память для хранения названий рецептов. Задание 1. Символ 13
D10013	WORD	Память для хранения названий рецептов. Задание 1. Символ 14
D10014	WORD	Память для хранения названий рецептов. Задание 1. Символ 15
D10015	WORD	Память для хранения названий рецептов. Задание 1. Символ 16
D10016	WORD	Память для хранения названий рецептов. Задание 1. Символ 17
D10017	WORD	Память для хранения названий рецептов. Задание 1. Символ 18
D10018	WORD	Память для хранения названий рецептов. Задание 1. Символ 19
D10019	WORD	Память для хранения названий рецептов. Задание 1. Символ 20
D10020	WORD	Память для хранения названий рецептов. Задание 1. Символ 21
D10021	WORD	Память для хранения названий рецептов. Задание 1. Символ 22
D10022	WORD	Память для хранения названий рецептов. Задание 1. Символ 23
D10023	WORD	Память для хранения названий рецептов. Задание 1. Символ 24
D10024	WORD	Память для хранения названий рецептов. Задание 1. Символ 25
D10025	WORD	Память для хранения названий рецептов. Задание 2. Символ 1
D10026	WORD	Память для хранения названий рецептов. Задание 2. Символ 2
D10027	WORD	Память для хранения названий рецептов. Задание 2. Символ 3
D10028	WORD	Память для хранения названий рецептов. Задание 2. Символ 4
D10029	WORD	Память для хранения названий рецептов. Задание 2. Символ 5
D10030	WORD	Память для хранения названий рецептов. Задание 2. Символ 6
D10031	WORD	Память для хранения названий рецептов. Задание 2. Символ 7
D10032	WORD	Память для хранения названий рецептов. Задание 2. Символ 8
D10033	WORD	Память для хранения названий рецептов. Задание 2. Символ 9
D10034	WORD	Память для хранения названий рецептов. Задание 2. Символ 10
D10035	WORD	Память для хранения названий рецептов. Задание 2. Символ 11
D10036	WORD	Память для хранения названий рецептов. Задание 2. Символ 12
D10037	WORD	Память для хранения названий рецептов. Задание 2. Символ 13
D10038	WORD	Память для хранения названий рецептов. Задание 2. Символ 14
D10039	WORD	Память для хранения названий рецептов. Задание 2. Символ 15
D10040	WORD	Память для хранения названий рецептов. Задание 2. Символ 16
D10041	WORD	Память для хранения названий рецептов. Задание 2. Символ 17
D10042	WORD	Память для хранения названий рецептов. Задание 2. Символ 18
D10043	WORD	Память для хранения названий рецептов. Задание 2. Символ 19
D10044	WORD	Память для хранения названий рецептов. Задание 2. Символ 20
D10045	WORD	Память для хранения названий рецептов. Задание 2. Символ 21
D10046	WORD	Память для хранения названий рецептов. Задание 2. Символ 22
D10047	WORD	Память для хранения названий рецептов. Задание 2. Символ 23
D10048	WORD	Память для хранения названий рецептов. Задание 2. Символ 24
D10049	WORD	Память для хранения названий рецептов. Задание 2. Символ 25
D10050	WORD	Память для хранения названий рецептов. Задание 3. Символ 1
D10051	WORD	Память для хранения названий рецептов. Задание 3. Символ 2
D10052	WORD	Память для хранения названий рецептов. Задание 3. Символ 3
D10053	WORD	Память для хранения названий рецептов. Задание 3. Символ 4
D10054	WORD	Память для хранения названий рецептов. Задание 3. Символ 5
D10055	WORD	Память для хранения названий рецептов. Задание 3. Символ 6
D10056	WORD	Память для хранения названий рецептов. Задание 3. Символ 7
D10057	WORD	Память для хранения названий рецептов. Задание 3. Символ 8
D10058	WORD	Память для хранения названий рецептов. Задание 3. Символ 9
D10059	WORD	Память для хранения названий рецептов. Задание 3. Символ 10
D10060	WORD	Память для хранения названий рецептов. Задание 3. Символ 11
D10061	WORD	Память для хранения названий рецептов. Задание 3. Символ 12
D10062	WORD	Память для хранения названий рецептов. Задание 3. Символ 13
D10063	WORD	Память для хранения названий рецептов. Задание 3. Символ 14
D10064	WORD	Память для хранения названий рецептов. Задание 3. Символ 15
D10065	WORD	Память для хранения названий рецептов. Задание 3. Символ 16
D10066	WORD	Память для хранения названий рецептов. Задание 3. Символ 17
D10067	WORD	Память для хранения названий рецептов. Задание 3. Символ 18
D10068	WORD	Память для хранения названий рецептов. Задание 3. Символ 19
D10069	WORD	Память для хранения названий рецептов. Задание 3. Символ 20
D10070	WORD	Память для хранения названий рецептов. Задание 3. Символ 21
D10071	WORD	Память для хранения названий рецептов. Задание 3. Символ 22
D10072	WORD	Память для хранения названий рецептов. Задание 3. Символ 23
D10073	WORD	Память для хранения названий рецептов. Задание 3. Символ 24
D10074	WORD	Память для хранения названий рецептов. Задание 3. Символ 25
D10075	WORD	Память для хранения названий рецептов. Задание 4. Символ 1
D10076	WORD	Память для хранения названий рецептов. Задание 4. Символ 2
D10077	WORD	Память для хранения названий рецептов. Задание 4. Символ 3
D10078	WORD	Память для хранения названий рецептов. Задание 4. Символ 4
D10079	WORD	Память для хранения названий рецептов. Задание 4. Символ 5
D10080	WORD	Память для хранения названий рецептов. Задание 4. Символ 6
D10081	WORD	Память для хранения названий рецептов. Задание 4. Символ 7
D10082	WORD	Память для хранения названий рецептов. Задание 4. Символ 8
D10083	WORD	Память для хранения названий рецептов. Задание 4. Символ 9
D10084	WORD	Память для хранения названий рецептов. Задание 4. Символ 10
D10085	WORD	Память для хранения названий рецептов. Задание 4. Символ 11
D10086	WORD	Память для хранения названий рецептов. Задание 4. Символ 12
D10087	WORD	Память для хранения названий рецептов. Задание 4. Символ 13
D10088	WORD	Память для хранения названий рецептов. Задание 4. Символ 14
D10089	WORD	Память для хранения названий рецептов. Задание 4. Символ 15
D10090	WORD	Память для хранения названий рецептов. Задание 4. Символ 16
D10091	WORD	Память для хранения названий рецептов. Задание 4. Символ 17
D10092	WORD	Память для хранения названий рецептов. Задание 4. Символ 18
D10093	WORD	Память для хранения названий рецептов. Задание 4. Символ 19
D10094	WORD	Память для хранения названий рецептов. Задание 4. Символ 20
D10095	WORD	Память для хранения названий рецептов. Задание 4. Символ 21
D10096	WORD	Память для хранения названий рецептов. Задание 4. Символ 22
D10097	WORD	Память для хранения названий рецептов. Задание 4. Символ 23
D10098	WORD	Память для хранения названий рецептов. Задание 4. Символ 24
D10099	WORD	Память для хранения названий рецептов. Задание 4. Символ 25
D10100	WORD	Память для хранения названий рецептов. Задание 5. Символ 1
D10101	WORD	Память для хранения названий рецептов. Задание 5. Символ 2
D10102	WORD	Память для хранения названий рецептов. Задание 5. Символ 3
D10103	WORD	Память для хранения названий рецептов. Задание 5. Символ 4
D10104	WORD	Память для хранения названий рецептов. Задание 5. Символ 5
D10105	WORD	Память для хранения названий рецептов. Задание 5. Символ 6
D10106	WORD	Память для хранения названий рецептов. Задание 5. Символ 7
D10107	WORD	Память для хранения названий рецептов. Задание 5. Символ 8
D10108	WORD	Память для хранения названий рецептов. Задание 5. Символ 9
D10109	WORD	Память для хранения названий рецептов. Задание 5. Символ 10
D10110	WORD	Память для хранения названий рецептов. Задание 5. Символ 11
D10111	WORD	Память для хранения названий рецептов. Задание 5. Символ 12
D10112	WORD	Память для хранения названий рецептов. Задание 5. Символ 13
D10113	WORD	Память для хранения названий рецептов. Задание 5. Символ 14
D10114	WORD	Память для хранения названий рецептов. Задание 5. Символ 15
D10115	WORD	Память для хранения названий рецептов. Задание 5. Символ 16
D10116	WORD	Память для хранения названий рецептов. Задание 5. Символ 17
D10117	WORD	Память для хранения названий рецептов. Задание 5. Символ 18
D10118	WORD	Память для хранения названий рецептов. Задание 5. Символ 19
D10119	WORD	Память для хранения названий рецептов. Задание 5. Символ 20
D10120	WORD	Память для хранения названий рецептов. Задание 5. Символ 21
D10121	WORD	Память для хранения названий рецептов. Задание 5. Символ 22
D10122	WORD	Память для хранения названий рецептов. Задание 5. Символ 23
D10123	WORD	Память для хранения названий рецептов. Задание 5. Символ 24
D10124	WORD	Память для хранения названий рецептов. Задание 5. Символ 25
D10125	WORD	Память для хранения названий рецептов. Задание 6. Символ 1
D10126	WORD	Память для хранения названий рецептов. Задание 6. Символ 2
D10127	WORD	Память для хранения названий рецептов. Задание 6. Символ 3
D10128	WORD	Память для хранения названий рецептов. Задание 6. Символ 4
D10129	WORD	Память для хранения названий рецептов. Задание 6. Символ 5
D10130	WORD	Память для хранения названий рецептов. Задание 6. Символ 6
D10131	WORD	Память для хранения названий рецептов. Задание 6. Символ 7
D10132	WORD	Память для хранения названий рецептов. Задание 6. Символ 8
D10133	WORD	Память для хранения названий рецептов. Задание 6. Символ 9
D10134	WORD	Память для хранения названий рецептов. Задание 6. Символ 10
D10135	WORD	Память для хранения названий рецептов. Задание 6. Символ 11
D10136	WORD	Память для хранения названий рецептов. Задание 6. Символ 12
D10137	WORD	Память для хранения названий рецептов. Задание 6. Символ 13
D10138	WORD	Память для хранения названий рецептов. Задание 6. Символ 14
D10139	WORD	Память для хранения названий рецептов. Задание 6. Символ 15
D10140	WORD	Память для хранения названий рецептов. Задание 6. Символ 16
D10141	WORD	Память для хранения названий рецептов. Задание 6. Символ 17
D10142	WORD	Память для хранения названий рецептов. Задание 6. Символ 18
D10143	WORD	Память для хранения названий рецептов. Задание 6. Символ 19
D10144	WORD	Память для хранения названий рецептов. Задание 6. Символ 20
D10145	WORD	Память для хранения названий рецептов. Задание 6. Символ 21
D10146	WORD	Память для хранения названий рецептов. Задание 6. Символ 22
D10147	WORD	Память для хранения названий рецептов. Задание 6. Символ 23
D10148	WORD	Память для хранения названий рецептов. Задание 6. Символ 24
D10149	WORD	Память для хранения названий рецептов. Задание 6. Символ 25
D10150	WORD	Память для хранения названий рецептов. Задание 7. Символ 1
D10151	WORD	Память для хранения названий рецептов. Задание 7. Символ 2
D10152	WORD	Память для хранения названий рецептов. Задание 7. Символ 3
D10153	WORD	Память для хранения названий рецептов. Задание 7. Символ 4
D10154	WORD	Память для хранения названий рецептов. Задание 7. Символ 5
D10155	WORD	Память для хранения названий рецептов. Задание 7. Символ 6
D10156	WORD	Память для хранения названий рецептов. Задание 7. Символ 7
D10157	WORD	Память для хранения названий рецептов. Задание 7. Символ 8
D10158	WORD	Память для хранения названий рецептов. Задание 7. Символ 9
D10159	WORD	Память для хранения названий рецептов. Задание 7. Символ 10
D10160	WORD	Память для хранения названий рецептов. Задание 7. Символ 11
D10161	WORD	Память для хранения названий рецептов. Задание 7. Символ 12
D10162	WORD	Память для хранения названий рецептов. Задание 7. Символ 13
D10163	WORD	Память для хранения названий рецептов. Задание 7. Символ 14
D10164	WORD	Память для хранения названий рецептов. Задание 7. Символ 15
D10165	WORD	Память для хранения названий рецептов. Задание 7. Символ 16
D10166	WORD	Память для хранения названий рецептов. Задание 7. Символ 17
D10167	WORD	Память для хранения названий рецептов. Задание 7. Символ 18
D10168	WORD	Память для хранения названий рецептов. Задание 7. Символ 19
D10169	WORD	Память для хранения названий рецептов. Задание 7. Символ 20
D10170	WORD	Память для хранения названий рецептов. Задание 7. Символ 21
D10171	WORD	Память для хранения названий рецептов. Задание 7. Символ 22
D10172	WORD	Память для хранения названий рецептов. Задание 7. Символ 23
D10173	WORD	Память для хранения названий рецептов. Задание 7. Символ 24
D10174	WORD	Память для хранения названий рецептов. Задание 7. Символ 25
D10175	WORD	Память для хранения названий рецептов. Задание 8. Символ 1
D10176	WORD	Память для хранения названий рецептов. Задание 8. Символ 2
D10177	WORD	Память для хранения названий рецептов. Задание 8. Символ 3
D10178	WORD	Память для хранения названий рецептов. Задание 8. Символ 4
D10179	WORD	Память для хранения названий рецептов. Задание 8. Символ 5
D10180	WORD	Память для хранения названий рецептов. Задание 8. Символ 6
D10181	WORD	Память для хранения названий рецептов. Задание 8. Символ 7
D10182	WORD	Память для хранения названий рецептов. Задание 8. Символ 8
D10183	WORD	Память для хранения названий рецептов. Задание 8. Символ 9
D10184	WORD	Память для хранения названий рецептов. Задание 8. Символ 10
D10185	WORD	Память для хранения названий рецептов. Задание 8. Символ 11
D10186	WORD	Память для хранения названий рецептов. Задание 8. Символ 12
D10187	WORD	Память для хранения названий рецептов. Задание 8. Символ 13
D10188	WORD	Память для хранения названий рецептов. Задание 8. Символ 14
D10189	WORD	Память для хранения названий рецептов. Задание 8. Символ 15
D10190	WORD	Память для хранения названий рецептов. Задание 8. Символ 16
D10191	WORD	Память для хранения названий рецептов. Задание 8. Символ 17
D10192	WORD	Память для хранения названий рецептов. Задание 8. Символ 18
D10193	WORD	Память для хранения названий рецептов. Задание 8. Символ 19
D10194	WORD	Память для хранения названий рецептов. Задание 8. Символ 20
D10195	WORD	Память для хранения названий рецептов. Задание 8. Символ 21
D10196	WORD	Память для хранения названий рецептов. Задание 8. Символ 22
D10197	WORD	Память для хранения названий рецептов. Задание 8. Символ 23
D10198	WORD	Память для хранения названий рецептов. Задание 8. Символ 24
D10199	WORD	Память для хранения названий рецептов. Задание 8. Символ 25
D10200	WORD	Память для хранения названий рецептов. Задание 9. Символ 1
D10201	WORD	Память для хранения названий рецептов. Задание 9. Символ 2
D10202	WORD	Память для хранения названий рецептов. Задание 9. Символ 3
D10203	WORD	Память для хранения названий рецептов. Задание 9. Символ 4
D10204	WORD	Память для хранения названий рецептов. Задание 9. Символ 5
D10205	WORD	Память для хранения названий рецептов. Задание 9. Символ 6
D10206	WORD	Память для хранения названий рецептов. Задание 9. Символ 7
D10207	WORD	Память для хранения названий рецептов. Задание 9. Символ 8
D10208	WORD	Память для хранения названий рецептов. Задание 9. Символ 9
D10209	WORD	Память для хранения названий рецептов. Задание 9. Символ 10
D10210	WORD	Память для хранения названий рецептов. Задание 9. Символ 11
D10211	WORD	Память для хранения названий рецептов. Задание 9. Символ 12
D10212	WORD	Память для хранения названий рецептов. Задание 9. Символ 13
D10213	WORD	Память для хранения названий рецептов. Задание 9. Символ 14
D10214	WORD	Память для хранения названий рецептов. Задание 9. Символ 15
D10215	WORD	Память для хранения названий рецептов. Задание 9. Символ 16
D10216	WORD	Память для хранения названий рецептов. Задание 9. Символ 17
D10217	WORD	Память для хранения названий рецептов. Задание 9. Символ 18
D10218	WORD	Память для хранения названий рецептов. Задание 9. Символ 19
D10219	WORD	Память для хранения названий рецептов. Задание 9. Символ 20
D10220	WORD	Память для хранения названий рецептов. Задание 9. Символ 21
D10221	WORD	Память для хранения названий рецептов. Задание 9. Символ 22
D10222	WORD	Память для хранения названий рецептов. Задание 9. Символ 23
D10223	WORD	Память для хранения названий рецептов. Задание 9. Символ 24
D10224	WORD	Память для хранения названий рецептов. Задание 9. Символ 25
D10225	WORD	Память для хранения названий рецептов. Задание 10. Символ 1
D10226	WORD	Память для хранения названий рецептов. Задание 10. Символ 2
D10227	WORD	Память для хранения названий рецептов. Задание 10. Символ 3
D10228	WORD	Память для хранения названий рецептов. Задание 10. Символ 4
D10229	WORD	Память для хранения названий рецептов. Задание 10. Символ 5
D10230	WORD	Память для хранения названий рецептов. Задание 10. Символ 6
D10231	WORD	Память для хранения названий рецептов. Задание 10. Символ 7
D10232	WORD	Память для хранения названий рецептов. Задание 10. Символ 8
D10233	WORD	Память для хранения названий рецептов. Задание 10. Символ 9
D10234	WORD	Память для хранения названий рецептов. Задание 10. Символ 10
D10235	WORD	Память для хранения названий рецептов. Задание 10. Символ 11
D10236	WORD	Память для хранения названий рецептов. Задание 10. Символ 12
D10237	WORD	Память для хранения названий рецептов. Задание 10. Символ 13
D10238	WORD	Память для хранения названий рецептов. Задание 10. Символ 14
D10239	WORD	Память для хранения названий рецептов. Задание 10. Символ 15
D10240	WORD	Память для хранения названий рецептов. Задание 10. Символ 16
D10241	WORD	Память для хранения названий рецептов. Задание 10. Символ 17
D10242	WORD	Память для хранения названий рецептов. Задание 10. Символ 18
D10243	WORD	Память для хранения названий рецептов. Задание 10. Символ 19
D10244	WORD	Память для хранения названий рецептов. Задание 10. Символ 20
D10245	WORD	Память для хранения названий рецептов. Задание 10. Символ 21
D10246	WORD	Память для хранения названий рецептов. Задание 10. Символ 22
D10247	WORD	Память для хранения названий рецептов. Задание 10. Символ 23
D10248	WORD	Память для хранения названий рецептов. Задание 10. Символ 24
D10249	WORD	Память для хранения названий рецептов. Задание 10. Символ 25
D10250	WORD	Память для хранения названий рецептов. Задание 11. Символ 1
D10251	WORD	Память для хранения названий рецептов. Задание 11. Символ 2
D10252	WORD	Память для хранения названий рецептов. Задание 11. Символ 3
D10253	WORD	Память для хранения названий рецептов. Задание 11. Символ 4
D10254	WORD	Память для хранения названий рецептов. Задание 11. Символ 5
D10255	WORD	Память для хранения названий рецептов. Задание 11. Символ 6
D10256	WORD	Память для хранения названий рецептов. Задание 11. Символ 7
D10257	WORD	Память для хранения названий рецептов. Задание 11. Символ 8
D10258	WORD	Память для хранения названий рецептов. Задание 11. Символ 9
D10259	WORD	Память для хранения названий рецептов. Задание 11. Символ 10
D10260	WORD	Память для хранения названий рецептов. Задание 11. Символ 11
D10261	WORD	Память для хранения названий рецептов. Задание 11. Символ 12
D10262	WORD	Память для хранения названий рецептов. Задание 11. Символ 13
D10263	WORD	Память для хранения названий рецептов. Задание 11. Символ 14
D10264	WORD	Память для хранения названий рецептов. Задание 11. Символ 15
D10265	WORD	Память для хранения названий рецептов. Задание 11. Символ 16
D10266	WORD	Память для хранения названий рецептов. Задание 11. Символ 17
D10267	WORD	Память для хранения названий рецептов. Задание 11. Символ 18
D10268	WORD	Память для хранения названий рецептов. Задание 11. Символ 19
D10269	WORD	Память для хранения названий рецептов. Задание 11. Символ 20
D10270	WORD	Память для хранения названий рецептов. Задание 11. Символ 21
D10271	WORD	Память для хранения названий рецептов. Задание 11. Символ 22
D10272	WORD	Память для хранения названий рецептов. Задание 11. Символ 23
D10273	WORD	Память для хранения названий рецептов. Задание 11. Символ 24
D10274	WORD	Память для хранения названий рецептов. Задание 11. Символ 25
D10275	WORD	Память для хранения названий рецептов. Задание 12. Символ 1
D10276	WORD	Память для хранения названий рецептов. Задание 12. Символ 2
D10277	WORD	Память для хранения названий рецептов. Задание 12. Символ 3
D10278	WORD	Память для хранения названий рецептов. Задание 12. Символ 4
D10279	WORD	Память для хранения названий рецептов. Задание 12. Символ 5
D10280	WORD	Память для хранения названий рецептов. Задание 12. Символ 6
D10281	WORD	Память для хранения названий рецептов. Задание 12. Символ 7
D10282	WORD	Память для хранения названий рецептов. Задание 12. Символ 8
D10283	WORD	Память для хранения названий рецептов. Задание 12. Символ 9
D10284	WORD	Память для хранения названий рецептов. Задание 12. Символ 10
D10285	WORD	Память для хранения названий рецептов. Задание 12. Символ 11
D10286	WORD	Память для хранения названий рецептов. Задание 12. Символ 12
D10287	WORD	Память для хранения названий рецептов. Задание 12. Символ 13
D10288	WORD	Память для хранения названий рецептов. Задание 12. Символ 14
D10289	WORD	Память для хранения названий рецептов. Задание 12. Символ 15
D10290	WORD	Память для хранения названий рецептов. Задание 12. Символ 16
D10291	WORD	Память для хранения названий рецептов. Задание 12. Символ 17
D10292	WORD	Память для хранения названий рецептов. Задание 12. Символ 18
D10293	WORD	Память для хранения названий рецептов. Задание 12. Символ 19
D10294	WORD	Память для хранения названий рецептов. Задание 12. Символ 20
D10295	WORD	Память для хранения названий рецептов. Задание 12. Символ 21
D10296	WORD	Память для хранения названий рецептов. Задание 12. Символ 22
D10297	WORD	Память для хранения названий рецептов. Задание 12. Символ 23
D10298	WORD	Память для хранения названий рецептов. Задание 12. Символ 24
D10299	WORD	Память для хранения названий рецептов. Задание 12. Символ 25
D10300	WORD	Память для хранения названий рецептов. Задание 13. Символ 1
D10301	WORD	Память для хранения названий рецептов. Задание 13. Символ 2
D10302	WORD	Память для хранения названий рецептов. Задание 13. Символ 3
D10303	WORD	Память для хранения названий рецептов. Задание 13. Символ 4
D10304	WORD	Память для хранения названий рецептов. Задание 13. Символ 5
D10305	WORD	Память для хранения названий рецептов. Задание 13. Символ 6
D10306	WORD	Память для хранения названий рецептов. Задание 13. Символ 7
D10307	WORD	Память для хранения названий рецептов. Задание 13. Символ 8
D10308	WORD	Память для хранения названий рецептов. Задание 13. Символ 9
D10309	WORD	Память для хранения названий рецептов. Задание 13. Символ 10
D10310	WORD	Память для хранения названий рецептов. Задание 13. Символ 11
D10311	WORD	Память для хранения названий рецептов. Задание 13. Символ 12
D10312	WORD	Память для хранения названий рецептов. Задание 13. Символ 13
D10313	WORD	Память для хранения названий рецептов. Задание 13. Символ 14
D10314	WORD	Память для хранения названий рецептов. Задание 13. Символ 15
D10315	WORD	Память для хранения названий рецептов. Задание 13. Символ 16
D10316	WORD	Память для хранения названий рецептов. Задание 13. Символ 17
D10317	WORD	Память для хранения названий рецептов. Задание 13. Символ 18
D10318	WORD	Память для хранения названий рецептов. Задание 13. Символ 19
D10319	WORD	Память для хранения названий рецептов. Задание 13. Символ 20
D10320	WORD	Память для хранения названий рецептов. Задание 13. Символ 21
D10321	WORD	Память для хранения названий рецептов. Задание 13. Символ 22
D10322	WORD	Память для хранения названий рецептов. Задание 13. Символ 23
D10323	WORD	Память для хранения названий рецептов. Задание 13. Символ 24
D10324	WORD	Память для хранения названий рецептов. Задание 13. Символ 25
D10325	WORD	Память для хранения названий рецептов. Задание 14. Символ 1
D10326	WORD	Память для хранения названий рецептов. Задание 14. Символ 2
D10327	WORD	Память для хранения названий рецептов. Задание 14. Символ 3
D10328	WORD	Память для хранения названий рецептов. Задание 14. Символ 4
D10329	WORD	Память для хранения названий рецептов. Задание 14. Символ 5
D10330	WORD	Память для хранения названий рецептов. Задание 14. Символ 6
D10331	WORD	Память для хранения названий рецептов. Задание 14. Символ 7
D10332	WORD	Память для хранения названий рецептов. Задание 14. Символ 8
D10333	WORD	Память для хранения названий рецептов. Задание 14. Символ 9
D10334	WORD	Память для хранения названий рецептов. Задание 14. Символ 10
D10335	WORD	Память для хранения названий рецептов. Задание 14. Символ 11
D10336	WORD	Память для хранения названий рецептов. Задание 14. Символ 12
D10337	WORD	Память для хранения названий рецептов. Задание 14. Символ 13
D10338	WORD	Память для хранения названий рецептов. Задание 14. Символ 14
D10339	WORD	Память для хранения названий рецептов. Задание 14. Символ 15
D10340	WORD	Память для хранения названий рецептов. Задание 14. Символ 16
D10341	WORD	Память для хранения названий рецептов. Задание 14. Символ 17
D10342	WORD	Память для хранения названий рецептов. Задание 14. Символ 18
D10343	WORD	Память для хранения названий рецептов. Задание 14. Символ 19
D10344	WORD	Память для хранения названий рецептов. Задание 14. Символ 20
D10345	WORD	Память для хранения названий рецептов. Задание 14. Символ 21
D10346	WORD	Память для хранения названий рецептов. Задание 14. Символ 22
D10347	WORD	Память для хранения названий рецептов. Задание 14. Символ 23
D10348	WORD	Память для хранения названий рецептов. Задание 14. Символ 24
D10349	WORD	Память для хранения названий рецептов. Задание 14. Символ 25
D10350	WORD	Память для хранения названий рецептов. Задание 15. Символ 1
D10351	WORD	Память для хранения названий рецептов. Задание 15. Символ 2
D10352	WORD	Память для хранения названий рецептов. Задание 15. Символ 3
D10353	WORD	Память для хранения названий рецептов. Задание 15. Символ 4
D10354	WORD	Память для хранения названий рецептов. Задание 15. Символ 5
D10355	WORD	Память для хранения названий рецептов. Задание 15. Символ 6
D10356	WORD	Память для хранения названий рецептов. Задание 15. Символ 7
D10357	WORD	Память для хранения названий рецептов. Задание 15. Символ 8
D10358	WORD	Память для хранения названий рецептов. Задание 15. Символ 9
D10359	WORD	Память для хранения названий рецептов. Задание 15. Символ 10
D10360	WORD	Память для хранения названий рецептов. Задание 15. Символ 11
D10361	WORD	Память для хранения названий рецептов. Задание 15. Символ 12
D10362	WORD	Память для хранения названий рецептов. Задание 15. Символ 13
D10363	WORD	Память для хранения названий рецептов. Задание 15. Символ 14
D10364	WORD	Память для хранения названий рецептов. Задание 15. Символ 15
D10365	WORD	Память для хранения названий рецептов. Задание 15. Символ 16
D10366	WORD	Память для хранения названий рецептов. Задание 15. Символ 17
D10367	WORD	Память для хранения названий рецептов. Задание 15. Символ 18
D10368	WORD	Память для хранения названий рецептов. Задание 15. Символ 19
D10369	WORD	Память для хранения названий рецептов. Задание 15. Символ 20
D10370	WORD	Память для хранения названий рецептов. Задание 15. Символ 21
D10371	WORD	Память для хранения названий рецептов. Задание 15. Символ 22
D10372	WORD	Память для хранения названий рецептов. Задание 15. Символ 23
D10373	WORD	Память для хранения названий рецептов. Задание 15. Символ 24
D10374	WORD	Память для хранения названий рецептов. Задание 15. Символ 25
D10375	WORD	Память для хранения названий рецептов. Задание 16. Символ 1
D10376	WORD	Память для хранения названий рецептов. Задание 16. Символ 2
D10377	WORD	Память для хранения названий рецептов. Задание 16. Символ 3
D10378	WORD	Память для хранения названий рецептов. Задание 16. Символ 4
D10379	WORD	Память для хранения названий рецептов. Задание 16. Символ 5
D10380	WORD	Память для хранения названий рецептов. Задание 16. Символ 6
D10381	WORD	Память для хранения названий рецептов. Задание 16. Символ 7
D10382	WORD	Память для хранения названий рецептов. Задание 16. Символ 8
D10383	WORD	Память для хранения названий рецептов. Задание 16. Символ 9
D10384	WORD	Память для хранения названий рецептов. Задание 16. Символ 10
D10385	WORD	Память для хранения названий рецептов. Задание 16. Символ 11
D10386	WORD	Память для хранения названий рецептов. Задание 16. Символ 12
D10387	WORD	Память для хранения названий рецептов. Задание 16. Символ 13
D10388	WORD	Память для хранения названий рецептов. Задание 16. Символ 14
D10389	WORD	Память для хранения названий рецептов. Задание 16. Символ 15
D10390	WORD	Память для хранения названий рецептов. Задание 16. Символ 16
D10391	WORD	Память для хранения названий рецептов. Задание 16. Символ 17
D10392	WORD	Память для хранения названий рецептов. Задание 16. Символ 18
D10393	WORD	Память для хранения названий рецептов. Задание 16. Символ 19
D10394	WORD	Память для хранения названий рецептов. Задание 16. Символ 20
D10395	WORD	Память для хранения названий рецептов. Задание 16. Символ 21
D10396	WORD	Память для хранения названий рецептов. Задание 16. Символ 22
D10397	WORD	Память для хранения названий рецептов. Задание 16. Символ 23
D10398	WORD	Память для хранения названий рецептов. Задание 16. Символ 24
D10399	WORD	Память для хранения названий рецептов. Задание 16. Символ 25
D10400	WORD	Память для хранения названий рецептов. Задание 17. Символ 1
D10401	WORD	Память для хранения названий рецептов. Задание 17. Символ 2
D10402	WORD	Память для хранения названий рецептов. Задание 17. Символ 3
D10403	WORD	Память для хранения названий рецептов. Задание 17. Символ 4
D10404	WORD	Память для хранения названий рецептов. Задание 17. Символ 5
D10405	WORD	Память для хранения названий рецептов. Задание 17. Символ 6
D10406	WORD	Память для хранения названий рецептов. Задание 17. Символ 7
D10407	WORD	Память для хранения названий рецептов. Задание 17. Символ 8
D10408	WORD	Память для хранения названий рецептов. Задание 17. Символ 9
D10409	WORD	Память для хранения названий рецептов. Задание 17. Символ 10
D10410	WORD	Память для хранения названий рецептов. Задание 17. Символ 11
D10411	WORD	Память для хранения названий рецептов. Задание 17. Символ 12
D10412	WORD	Память для хранения названий рецептов. Задание 17. Символ 13
D10413	WORD	Память для хранения названий рецептов. Задание 17. Символ 14
D10414	WORD	Память для хранения названий рецептов. Задание 17. Символ 15
D10415	WORD	Память для хранения названий рецептов. Задание 17. Символ 16
D10416	WORD	Память для хранения названий рецептов. Задание 17. Символ 17
D10417	WORD	Память для хранения названий рецептов. Задание 17. Символ 18
D10418	WORD	Память для хранения названий рецептов. Задание 17. Символ 19
D10419	WORD	Память для хранения названий рецептов. Задание 17. Символ 20
D10420	WORD	Память для хранения названий рецептов. Задание 17. Символ 21
D10421	WORD	Память для хранения названий рецептов. Задание 17. Символ 22
D10422	WORD	Память для хранения названий рецептов. Задание 17. Символ 23
D10423	WORD	Память для хранения названий рецептов. Задание 17. Символ 24
D10424	WORD	Память для хранения названий рецептов. Задание 17. Символ 25
D10425	WORD	Память для хранения названий рецептов. Задание 18. Символ 1
D10426	WORD	Память для хранения названий рецептов. Задание 18. Символ 2
D10427	WORD	Память для хранения названий рецептов. Задание 18. Символ 3
D10428	WORD	Память для хранения названий рецептов. Задание 18. Символ 4
D10429	WORD	Память для хранения названий рецептов. Задание 18. Символ 5
D10430	WORD	Память для хранения названий рецептов. Задание 18. Символ 6
D10431	WORD	Память для хранения названий рецептов. Задание 18. Символ 7
D10432	WORD	Память для хранения названий рецептов. Задание 18. Символ 8
D10433	WORD	Память для хранения названий рецептов. Задание 18. Символ 9
D10434	WORD	Память для хранения названий рецептов. Задание 18. Символ 10
D10435	WORD	Память для хранения названий рецептов. Задание 18. Символ 11
D10436	WORD	Память для хранения названий рецептов. Задание 18. Символ 12
D10437	WORD	Память для хранения названий рецептов. Задание 18. Символ 13
D10438	WORD	Память для хранения названий рецептов. Задание 18. Символ 14
D10439	WORD	Память для хранения названий рецептов. Задание 18. Символ 15
D10440	WORD	Память для хранения названий рецептов. Задание 18. Символ 16
D10441	WORD	Память для хранения названий рецептов. Задание 18. Символ 17
D10442	WORD	Память для хранения названий рецептов. Задание 18. Символ 18
D10443	WORD	Память для хранения названий рецептов. Задание 18. Символ 19
D10444	WORD	Память для хранения названий рецептов. Задание 18. Символ 20
D10445	WORD	Память для хранения названий рецептов. Задание 18. Символ 21
D10446	WORD	Память для хранения названий рецептов. Задание 18. Символ 22
D10447	WORD	Память для хранения названий рецептов. Задание 18. Символ 23
D10448	WORD	Память для хранения названий рецептов. Задание 18. Символ 24
D10449	WORD	Память для хранения названий рецептов. Задание 18. Символ 25
D10450	WORD	Память для хранения названий рецептов. Задание 19. Символ 1
D10451	WORD	Память для хранения названий рецептов. Задание 19. Символ 2
D10452	WORD	Память для хранения названий рецептов. Задание 19. Символ 3
D10453	WORD	Память для хранения названий рецептов. Задание 19. Символ 4
D10454	WORD	Память для хранения названий рецептов. Задание 19. Символ 5
D10455	WORD	Память для хранения названий рецептов. Задание 19. Символ 6
D10456	WORD	Память для хранения названий рецептов. Задание 19. Символ 7
D10457	WORD	Память для хранения названий рецептов. Задание 19. Символ 8
D10458	WORD	Память для хранения названий рецептов. Задание 19. Символ 9
D10459	WORD	Память для хранения названий рецептов. Задание 19. Символ 10
D10460	WORD	Память для хранения названий рецептов. Задание 19. Символ 11
D10461	WORD	Память для хранения названий рецептов. Задание 19. Символ 12
D10462	WORD	Память для хранения названий рецептов. Задание 19. Символ 13
D10463	WORD	Память для хранения названий рецептов. Задание 19. Символ 14
D10464	WORD	Память для хранения названий рецептов. Задание 19. Символ 15
D10465	WORD	Память для хранения названий рецептов. Задание 19. Символ 16
D10466	WORD	Память для хранения названий рецептов. Задание 19. Символ 17
D10467	WORD	Память для хранения названий рецептов. Задание 19. Символ 18
D10468	WORD	Память для хранения названий рецептов. Задание 19. Символ 19
D10469	WORD	Память для хранения названий рецептов. Задание 19. Символ 20
D10470	WORD	Память для хранения названий рецептов. Задание 19. Символ 21
D10471	WORD	Память для хранения названий рецептов. Задание 19. Символ 22
D10472	WORD	Память для хранения названий рецептов. Задание 19. Символ 23
D10473	WORD	Память для хранения названий рецептов. Задание 19. Символ 24
D10474	WORD	Память для хранения названий рецептов. Задание 19. Символ 25
D10475	WORD	Память для хранения названий рецептов. Задание 20. Символ 1
D10476	WORD	Память для хранения названий рецептов. Задание 20. Символ 2
D10477	WORD	Память для хранения названий рецептов. Задание 20. Символ 3
D10478	WORD	Память для хранения названий рецептов. Задание 20. Символ 4
D10479	WORD	Память для хранения названий рецептов. Задание 20. Символ 5
D10480	WORD	Память для хранения названий рецептов. Задание 20. Символ 6
D10481	WORD	Память для хранения названий рецептов. Задание 20. Символ 7
D10482	WORD	Память для хранения названий рецептов. Задание 20. Символ 8
D10483	WORD	Память для хранения названий рецептов. Задание 20. Символ 9
D10484	WORD	Память для хранения названий рецептов. Задание 20. Символ 10
D10485	WORD	Память для хранения названий рецептов. Задание 20. Символ 11
D10486	WORD	Память для хранения названий рецептов. Задание 20. Символ 12
D10487	WORD	Память для хранения названий рецептов. Задание 20. Символ 13
D10488	WORD	Память для хранения названий рецептов. Задание 20. Символ 14
D10489	WORD	Память для хранения названий рецептов. Задание 20. Символ 15
D10490	WORD	Память для хранения названий рецептов. Задание 20. Символ 16
D10491	WORD	Память для хранения названий рецептов. Задание 20. Символ 17
D10492	WORD	Память для хранения названий рецептов. Задание 20. Символ 18
D10493	WORD	Память для хранения названий рецептов. Задание 20. Символ 19
D10494	WORD	Память для хранения названий рецептов. Задание 20. Символ 20
D10495	WORD	Память для хранения названий рецептов. Задание 20. Символ 21
D10496	WORD	Память для хранения названий рецептов. Задание 20. Символ 22
D10497	WORD	Память для хранения названий рецептов. Задание 20. Символ 23
D10498	WORD	Память для хранения названий рецептов. Задание 20. Символ 24
D10499	WORD	Память для хранения названий рецептов. Задание 20. Символ 25
D10500	WORD	Память для хранения названий рецептов. Задание 21. Символ 1
D10501	WORD	Память для хранения названий рецептов. Задание 21. Символ 2
D10502	WORD	Память для хранения названий рецептов. Задание 21. Символ 3
D10503	WORD	Память для хранения названий рецептов. Задание 21. Символ 4
D10504	WORD	Память для хранения названий рецептов. Задание 21. Символ 5
D10505	WORD	Память для хранения названий рецептов. Задание 21. Символ 6
D10506	WORD	Память для хранения названий рецептов. Задание 21. Символ 7
D10507	WORD	Память для хранения названий рецептов. Задание 21. Символ 8
D10508	WORD	Память для хранения названий рецептов. Задание 21. Символ 9
D10509	WORD	Память для хранения названий рецептов. Задание 21. Символ 10
D10510	WORD	Память для хранения названий рецептов. Задание 21. Символ 11
D10511	WORD	Память для хранения названий рецептов. Задание 21. Символ 12
D10512	WORD	Память для хранения названий рецептов. Задание 21. Символ 13
D10513	WORD	Память для хранения названий рецептов. Задание 21. Символ 14
D10514	WORD	Память для хранения названий рецептов. Задание 21. Символ 15
D10515	WORD	Память для хранения названий рецептов. Задание 21. Символ 16
D10516	WORD	Память для хранения названий рецептов. Задание 21. Символ 17
D10517	WORD	Память для хранения названий рецептов. Задание 21. Символ 18
D10518	WORD	Память для хранения названий рецептов. Задание 21. Символ 19
D10519	WORD	Память для хранения названий рецептов. Задание 21. Символ 20
D10520	WORD	Память для хранения названий рецептов. Задание 21. Символ 21
D10521	WORD	Память для хранения названий рецептов. Задание 21. Символ 22
D10522	WORD	Память для хранения названий рецептов. Задание 21. Символ 23
D10523	WORD	Память для хранения названий рецептов. Задание 21. Символ 24
D10524	WORD	Память для хранения названий рецептов. Задание 21. Символ 25
D10525	WORD	Память для хранения названий рецептов. Задание 22. Символ 1
D10526	WORD	Память для хранения названий рецептов. Задание 22. Символ 2
D10527	WORD	Память для хранения названий рецептов. Задание 22. Символ 3
D10528	WORD	Память для хранения названий рецептов. Задание 22. Символ 4
D10529	WORD	Память для хранения названий рецептов. Задание 22. Символ 5
D10530	WORD	Память для хранения названий рецептов. Задание 22. Символ 6
D10531	WORD	Память для хранения названий рецептов. Задание 22. Символ 7
D10532	WORD	Память для хранения названий рецептов. Задание 22. Символ 8
D10533	WORD	Память для хранения названий рецептов. Задание 22. Символ 9
D10534	WORD	Память для хранения названий рецептов. Задание 22. Символ 10
D10535	WORD	Память для хранения названий рецептов. Задание 22. Символ 11
D10536	WORD	Память для хранения названий рецептов. Задание 22. Символ 12
D10537	WORD	Память для хранения названий рецептов. Задание 22. Символ 13
D10538	WORD	Память для хранения названий рецептов. Задание 22. Символ 14
D10539	WORD	Память для хранения названий рецептов. Задание 22. Символ 15
D10540	WORD	Память для хранения названий рецептов. Задание 22. Символ 16
D10541	WORD	Память для хранения названий рецептов. Задание 22. Символ 17
D10542	WORD	Память для хранения названий рецептов. Задание 22. Символ 18
D10543	WORD	Память для хранения названий рецептов. Задание 22. Символ 19
D10544	WORD	Память для хранения названий рецептов. Задание 22. Символ 20
D10545	WORD	Память для хранения названий рецептов. Задание 22. Символ 21
D10546	WORD	Память для хранения названий рецептов. Задание 22. Символ 22
D10547	WORD	Память для хранения названий рецептов. Задание 22. Символ 23
D10548	WORD	Память для хранения названий рецептов. Задание 22. Символ 24
D10549	WORD	Память для хранения названий рецептов. Задание 22. Символ 25
D10550	WORD	Память для хранения названий рецептов. Задание 23. Символ 1
D10551	WORD	Память для хранения названий рецептов. Задание 23. Символ 2
D10552	WORD	Память для хранения названий рецептов. Задание 23. Символ 3
D10553	WORD	Память для хранения названий рецептов. Задание 23. Символ 4
D10554	WORD	Память для хранения названий рецептов. Задание 23. Символ 5
D10555	WORD	Память для хранения названий рецептов. Задание 23. Символ 6
D10556	WORD	Память для хранения названий рецептов. Задание 23. Символ 7
D10557	WORD	Память для хранения названий рецептов. Задание 23. Символ 8
D10558	WORD	Память для хранения названий рецептов. Задание 23. Символ 9
D10559	WORD	Память для хранения названий рецептов. Задание 23. Символ 10
D10560	WORD	Память для хранения названий рецептов. Задание 23. Символ 11
D10561	WORD	Память для хранения названий рецептов. Задание 23. Символ 12
D10562	WORD	Память для хранения названий рецептов. Задание 23. Символ 13
D10563	WORD	Память для хранения названий рецептов. Задание 23. Символ 14
D10564	WORD	Память для хранения названий рецептов. Задание 23. Символ 15
D10565	WORD	Память для хранения названий рецептов. Задание 23. Символ 16
D10566	WORD	Память для хранения названий рецептов. Задание 23. Символ 17
D10567	WORD	Память для хранения названий рецептов. Задание 23. Символ 18
D10568	WORD	Память для хранения названий рецептов. Задание 23. Символ 19
D10569	WORD	Память для хранения названий рецептов. Задание 23. Символ 20
D10570	WORD	Память для хранения названий рецептов. Задание 23. Символ 21
D10571	WORD	Память для хранения названий рецептов. Задание 23. Символ 22
D10572	WORD	Память для хранения названий рецептов. Задание 23. Символ 23
D10573	WORD	Память для хранения названий рецептов. Задание 23. Символ 24
D10574	WORD	Память для хранения названий рецептов. Задание 23. Символ 25
D10575	WORD	Память для хранения названий рецептов. Задание 24. Символ 1
D10576	WORD	Память для хранения названий рецептов. Задание 24. Символ 2
D10577	WORD	Память для хранения названий рецептов. Задание 24. Символ 3
D10578	WORD	Память для хранения названий рецептов. Задание 24. Символ 4
D10579	WORD	Память для хранения названий рецептов. Задание 24. Символ 5
D10580	WORD	Память для хранения названий рецептов. Задание 24. Символ 6
D10581	WORD	Память для хранения названий рецептов. Задание 24. Символ 7
D10582	WORD	Память для хранения названий рецептов. Задание 24. Символ 8
D10583	WORD	Память для хранения названий рецептов. Задание 24. Символ 9
D10584	WORD	Память для хранения названий рецептов. Задание 24. Символ 10
D10585	WORD	Память для хранения названий рецептов. Задание 24. Символ 11
D10586	WORD	Память для хранения названий рецептов. Задание 24. Символ 12
D10587	WORD	Память для хранения названий рецептов. Задание 24. Символ 13
D10588	WORD	Память для хранения названий рецептов. Задание 24. Символ 14
D10589	WORD	Память для хранения названий рецептов. Задание 24. Символ 15
D10590	WORD	Память для хранения названий рецептов. Задание 24. Символ 16
D10591	WORD	Память для хранения названий рецептов. Задание 24. Символ 17
D10592	WORD	Память для хранения названий рецептов. Задание 24. Символ 18
D10593	WORD	Память для хранения названий рецептов. Задание 24. Символ 19
D10594	WORD	Память для хранения названий рецептов. Задание 24. Символ 20
D10595	WORD	Память для хранения названий рецептов. Задание 24. Символ 21
D10596	WORD	Память для хранения названий рецептов. Задание 24. Символ 22
D10597	WORD	Память для хранения названий рецептов. Задание 24. Символ 23
D10598	WORD	Память для хранения названий рецептов. Задание 24. Символ 24
D10599	WORD	Память для хранения названий рецептов. Задание 24. Символ 25
D10600	WORD	Память для хранения названий рецептов. Задание 25. Символ 1
D10601	WORD	Память для хранения названий рецептов. Задание 25. Символ 2
D10602	WORD	Память для хранения названий рецептов. Задание 25. Символ 3
D10603	WORD	Память для хранения названий рецептов. Задание 25. Символ 4
D10604	WORD	Память для хранения названий рецептов. Задание 25. Символ 5
D10605	WORD	Память для хранения названий рецептов. Задание 25. Символ 6
D10606	WORD	Память для хранения названий рецептов. Задание 25. Символ 7
D10607	WORD	Память для хранения названий рецептов. Задание 25. Символ 8
D10608	WORD	Память для хранения названий рецептов. Задание 25. Символ 9
D10609	WORD	Память для хранения названий рецептов. Задание 25. Символ 10
D10610	WORD	Память для хранения названий рецептов. Задание 25. Символ 11
D10611	WORD	Память для хранения названий рецептов. Задание 25. Символ 12
D10612	WORD	Память для хранения названий рецептов. Задание 25. Символ 13
D10613	WORD	Память для хранения названий рецептов. Задание 25. Символ 14
D10614	WORD	Память для хранения названий рецептов. Задание 25. Символ 15
D10615	WORD	Память для хранения названий рецептов. Задание 25. Символ 16
D10616	WORD	Память для хранения названий рецептов. Задание 25. Символ 17
D10617	WORD	Память для хранения названий рецептов. Задание 25. Символ 18
D10618	WORD	Память для хранения названий рецептов. Задание 25. Символ 19
D10619	WORD	Память для хранения названий рецептов. Задание 25. Символ 20
D10620	WORD	Память для хранения названий рецептов. Задание 25. Символ 21
D10621	WORD	Память для хранения названий рецептов. Задание 25. Символ 22
D10622	WORD	Память для хранения названий рецептов. Задание 25. Символ 23
D10623	WORD	Память для хранения названий рецептов. Задание 25. Символ 24
D10624	WORD	Память для хранения названий рецептов. Задание 25. Символ 25
D10625	WORD	Память для хранения названий рецептов. Задание 26. Символ 1
D10626	WORD	Память для хранения названий рецептов. Задание 26. Символ 2
D10627	WORD	Память для хранения названий рецептов. Задание 26. Символ 3
D10628	WORD	Память для хранения названий рецептов. Задание 26. Символ 4
D10629	WORD	Память для хранения названий рецептов. Задание 26. Символ 5
D10630	WORD	Память для хранения названий рецептов. Задание 26. Символ 6
D10631	WORD	Память для хранения названий рецептов. Задание 26. Символ 7
D10632	WORD	Память для хранения названий рецептов. Задание 26. Символ 8
D10633	WORD	Память для хранения названий рецептов. Задание 26. Символ 9
D10634	WORD	Память для хранения названий рецептов. Задание 26. Символ 10
D10635	WORD	Память для хранения названий рецептов. Задание 26. Символ 11
D10636	WORD	Память для хранения названий рецептов. Задание 26. Символ 12
D10637	WORD	Память для хранения названий рецептов. Задание 26. Символ 13
D10638	WORD	Память для хранения названий рецептов. Задание 26. Символ 14
D10639	WORD	Память для хранения названий рецептов. Задание 26. Символ 15
D10640	WORD	Память для хранения названий рецептов. Задание 26. Символ 16
D10641	WORD	Память для хранения названий рецептов. Задание 26. Символ 17
D10642	WORD	Память для хранения названий рецептов. Задание 26. Символ 18
D10643	WORD	Память для хранения названий рецептов. Задание 26. Символ 19
D10644	WORD	Память для хранения названий рецептов. Задание 26. Символ 20
D10645	WORD	Память для хранения названий рецептов. Задание 26. Символ 21
D10646	WORD	Память для хранения названий рецептов. Задание 26. Символ 22
D10647	WORD	Память для хранения названий рецептов. Задание 26. Символ 23
D10648	WORD	Память для хранения названий рецептов. Задание 26. Символ 24
D10649	WORD	Память для хранения названий рецептов. Задание 26. Символ 25
D10650	WORD	Память для хранения названий рецептов. Задание 27. Символ 1
D10651	WORD	Память для хранения названий рецептов. Задание 27. Символ 2
D10652	WORD	Память для хранения названий рецептов. Задание 27. Символ 3
D10653	WORD	Память для хранения названий рецептов. Задание 27. Символ 4
D10654	WORD	Память для хранения названий рецептов. Задание 27. Символ 5
D10655	WORD	Память для хранения названий рецептов. Задание 27. Символ 6
D10656	WORD	Память для хранения названий рецептов. Задание 27. Символ 7
D10657	WORD	Память для хранения названий рецептов. Задание 27. Символ 8
D10658	WORD	Память для хранения названий рецептов. Задание 27. Символ 9
D10659	WORD	Память для хранения названий рецептов. Задание 27. Символ 10
D10660	WORD	Память для хранения названий рецептов. Задание 27. Символ 11
D10661	WORD	Память для хранения названий рецептов. Задание 27. Символ 12
D10662	WORD	Память для хранения названий рецептов. Задание 27. Символ 13
D10663	WORD	Память для хранения названий рецептов. Задание 27. Символ 14
D10664	WORD	Память для хранения названий рецептов. Задание 27. Символ 15
D10665	WORD	Память для хранения названий рецептов. Задание 27. Символ 16
D10666	WORD	Память для хранения названий рецептов. Задание 27. Символ 17
D10667	WORD	Память для хранения названий рецептов. Задание 27. Символ 18
D10668	WORD	Память для хранения названий рецептов. Задание 27. Символ 19
D10669	WORD	Память для хранения названий рецептов. Задание 27. Символ 20
D10670	WORD	Память для хранения названий рецептов. Задание 27. Символ 21
D10671	WORD	Память для хранения названий рецептов. Задание 27. Символ 22
D10672	WORD	Память для хранения названий рецептов. Задание 27. Символ 23
D10673	WORD	Память для хранения названий рецептов. Задание 27. Символ 24
D10674	WORD	Память для хранения названий рецептов. Задание 27. Символ 25
D10675	WORD	Память для хранения названий рецептов. Задание 28. Символ 1
D10676	WORD	Память для хранения названий рецептов. Задание 28. Символ 2
D10677	WORD	Память для хранения названий рецептов. Задание 28. Символ 3
D10678	WORD	Память для хранения названий рецептов. Задание 28. Символ 4
D10679	WORD	Память для хранения названий рецептов. Задание 28. Символ 5
D10680	WORD	Память для хранения названий рецептов. Задание 28. Символ 6
D10681	WORD	Память для хранения названий рецептов. Задание 28. Символ 7
D10682	WORD	Память для хранения названий рецептов. Задание 28. Символ 8
D10683	WORD	Память для хранения названий рецептов. Задание 28. Символ 9
D10684	WORD	Память для хранения названий рецептов. Задание 28. Символ 10
D10685	WORD	Память для хранения названий рецептов. Задание 28. Символ 11
D10686	WORD	Память для хранения названий рецептов. Задание 28. Символ 12
D10687	WORD	Память для хранения названий рецептов. Задание 28. Символ 13
D10688	WORD	Память для хранения названий рецептов. Задание 28. Символ 14
D10689	WORD	Память для хранения названий рецептов. Задание 28. Символ 15
D10690	WORD	Память для хранения названий рецептов. Задание 28. Символ 16
D10691	WORD	Память для хранения названий рецептов. Задание 28. Символ 17
D10692	WORD	Память для хранения названий рецептов. Задание 28. Символ 18
D10693	WORD	Память для хранения названий рецептов. Задание 28. Символ 19
D10694	WORD	Память для хранения названий рецептов. Задание 28. Символ 20
D10695	WORD	Память для хранения названий рецептов. Задание 28. Символ 21
D10696	WORD	Память для хранения названий рецептов. Задание 28. Символ 22
D10697	WORD	Память для хранения названий рецептов. Задание 28. Символ 23
D10698	WORD	Память для хранения названий рецептов. Задание 28. Символ 24
D10699	WORD	Память для хранения названий рецептов. Задание 28. Символ 25
D10700	WORD	Память для хранения названий рецептов. Задание 29. Символ 1
D10701	WORD	Память для хранения названий рецептов. Задание 29. Символ 2
D10702	WORD	Память для хранения названий рецептов. Задание 29. Символ 3
D10703	WORD	Память для хранения названий рецептов. Задание 29. Символ 4
D10704	WORD	Память для хранения названий рецептов. Задание 29. Символ 5
D10705	WORD	Память для хранения названий рецептов. Задание 29. Символ 6
D10706	WORD	Память для хранения названий рецептов. Задание 29. Символ 7
D10707	WORD	Память для хранения названий рецептов. Задание 29. Символ 8
D10708	WORD	Память для хранения названий рецептов. Задание 29. Символ 9
D10709	WORD	Память для хранения названий рецептов. Задание 29. Символ 10
D10710	WORD	Память для хранения названий рецептов. Задание 29. Символ 11
D10711	WORD	Память для хранения названий рецептов. Задание 29. Символ 12
D10712	WORD	Память для хранения названий рецептов. Задание 29. Символ 13
D10713	WORD	Память для хранения названий рецептов. Задание 29. Символ 14
D10714	WORD	Память для хранения названий рецептов. Задание 29. Символ 15
D10715	WORD	Память для хранения названий рецептов. Задание 29. Символ 16
D10716	WORD	Память для хранения названий рецептов. Задание 29. Символ 17
D10717	WORD	Память для хранения названий рецептов. Задание 29. Символ 18
D10718	WORD	Память для хранения названий рецептов. Задание 29. Символ 19
D10719	WORD	Память для хранения названий рецептов. Задание 29. Символ 20
D10720	WORD	Память для хранения названий рецептов. Задание 29. Символ 21
D10721	WORD	Память для хранения названий рецептов. Задание 29. Символ 22
D10722	WORD	Память для хранения названий рецептов. Задание 29. Символ 23
D10723	WORD	Память для хранения названий рецептов. Задание 29. Символ 24
D10724	WORD	Память для хранения названий рецептов. Задание 29. Символ 25
D10725	WORD	Память для хранения названий рецептов. Задание 30. Символ 1
D10726	WORD	Память для хранения названий рецептов. Задание 30. Символ 2
D10727	WORD	Память для хранения названий рецептов. Задание 30. Символ 3
D10728	WORD	Память для хранения названий рецептов. Задание 30. Символ 4
D10729	WORD	Память для хранения названий рецептов. Задание 30. Символ 5
D10730	WORD	Память для хранения названий рецептов. Задание 30. Символ 6
D10731	WORD	Память для хранения названий рецептов. Задание 30. Символ 7
D10732	WORD	Память для хранения названий рецептов. Задание 30. Символ 8
D10733	WORD	Память для хранения названий рецептов. Задание 30. Символ 9
D10734	WORD	Память для хранения названий рецептов. Задание 30. Символ 10
D10735	WORD	Память для хранения названий рецептов. Задание 30. Символ 11
D10736	WORD	Память для хранения названий рецептов. Задание 30. Символ 12
D10737	WORD	Память для хранения названий рецептов. Задание 30. Символ 13
D10738	WORD	Память для хранения названий рецептов. Задание 30. Символ 14
D10739	WORD	Память для хранения названий рецептов. Задание 30. Символ 15
D10740	WORD	Память для хранения названий рецептов. Задание 30. Символ 16
D10741	WORD	Память для хранения названий рецептов. Задание 30. Символ 17
D10742	WORD	Память для хранения названий рецептов. Задание 30. Символ 18
D10743	WORD	Память для хранения названий рецептов. Задание 30. Символ 19
D10744	WORD	Память для хранения названий рецептов. Задание 30. Символ 20
D10745	WORD	Память для хранения названий рецептов. Задание 30. Символ 21
D10746	WORD	Память для хранения названий рецептов. Задание 30. Символ 22
D10747	WORD	Память для хранения названий рецептов. Задание 30. Символ 23
D10748	WORD	Память для хранения названий рецептов. Задание 30. Символ 24
D10749	WORD	Память для хранения названий рецептов. Задание 30. Символ 25
D10750	WORD	Память для хранения названий рецептов. Задание 31. Символ 1
D10751	WORD	Память для хранения названий рецептов. Задание 31. Символ 2
D10752	WORD	Память для хранения названий рецептов. Задание 31. Символ 3
D10753	WORD	Память для хранения названий рецептов. Задание 31. Символ 4
D10754	WORD	Память для хранения названий рецептов. Задание 31. Символ 5
D10755	WORD	Память для хранения названий рецептов. Задание 31. Символ 6
D10756	WORD	Память для хранения названий рецептов. Задание 31. Символ 7
D10757	WORD	Память для хранения названий рецептов. Задание 31. Символ 8
D10758	WORD	Память для хранения названий рецептов. Задание 31. Символ 9
D10759	WORD	Память для хранения названий рецептов. Задание 31. Символ 10
D10760	WORD	Память для хранения названий рецептов. Задание 31. Символ 11
D10761	WORD	Память для хранения названий рецептов. Задание 31. Символ 12
D10762	WORD	Память для хранения названий рецептов. Задание 31. Символ 13
D10763	WORD	Память для хранения названий рецептов. Задание 31. Символ 14
D10764	WORD	Память для хранения названий рецептов. Задание 31. Символ 15
D10765	WORD	Память для хранения названий рецептов. Задание 31. Символ 16
D10766	WORD	Память для хранения названий рецептов. Задание 31. Символ 17
D10767	WORD	Память для хранения названий рецептов. Задание 31. Символ 18
D10768	WORD	Память для хранения названий рецептов. Задание 31. Символ 19
D10769	WORD	Память для хранения названий рецептов. Задание 31. Символ 20
D10770	WORD	Память для хранения названий рецептов. Задание 31. Символ 21
D10771	WORD	Память для хранения названий рецептов. Задание 31. Символ 22
D10772	WORD	Память для хранения названий рецептов. Задание 31. Символ 23
D10773	WORD	Память для хранения названий рецептов. Задание 31. Символ 24
D10774	WORD	Память для хранения названий рецептов. Задание 31. Символ 25
D10775	WORD	Память для хранения названий рецептов. Задание 32. Символ 1
D10776	WORD	Память для хранения названий рецептов. Задание 32. Символ 2
D10777	WORD	Память для хранения названий рецептов. Задание 32. Символ 3
D10778	WORD	Память для хранения названий рецептов. Задание 32. Символ 4
D10779	WORD	Память для хранения названий рецептов. Задание 32. Символ 5
D10780	WORD	Память для хранения названий рецептов. Задание 32. Символ 6
D10781	WORD	Память для хранения названий рецептов. Задание 32. Символ 7
D10782	WORD	Память для хранения названий рецептов. Задание 32. Символ 8
D10783	WORD	Память для хранения названий рецептов. Задание 32. Символ 9
D10784	WORD	Память для хранения названий рецептов. Задание 32. Символ 10
D10785	WORD	Память для хранения названий рецептов. Задание 32. Символ 11
D10786	WORD	Память для хранения названий рецептов. Задание 32. Символ 12
D10787	WORD	Память для хранения названий рецептов. Задание 32. Символ 13
D10788	WORD	Память для хранения названий рецептов. Задание 32. Символ 14
D10789	WORD	Память для хранения названий рецептов. Задание 32. Символ 15
D10790	WORD	Память для хранения названий рецептов. Задание 32. Символ 16
D10791	WORD	Память для хранения названий рецептов. Задание 32. Символ 17
D10792	WORD	Память для хранения названий рецептов. Задание 32. Символ 18
D10793	WORD	Память для хранения названий рецептов. Задание 32. Символ 19
D10794	WORD	Память для хранения названий рецептов. Задание 32. Символ 20
D10795	WORD	Память для хранения названий рецептов. Задание 32. Символ 21
D10796	WORD	Память для хранения названий рецептов. Задание 32. Символ 22
D10797	WORD	Память для хранения названий рецептов. Задание 32. Символ 23
D10798	WORD	Память для хранения названий рецептов. Задание 32. Символ 24
D10799	WORD	Память для хранения названий рецептов. Задание 32. Символ 25
D10800	WORD	Память для хранения названий рецептов. Задание 33. Символ 1
D10801	WORD	Память для хранения названий рецептов. Задание 33. Символ 2
D10802	WORD	Память для хранения названий рецептов. Задание 33. Символ 3
D10803	WORD	Память для хранения названий рецептов. Задание 33. Символ 4
D10804	WORD	Память для хранения названий рецептов. Задание 33. Символ 5
D10805	WORD	Память для хранения названий рецептов. Задание 33. Символ 6
D10806	WORD	Память для хранения названий рецептов. Задание 33. Символ 7
D10807	WORD	Память для хранения названий рецептов. Задание 33. Символ 8
D10808	WORD	Память для хранения названий рецептов. Задание 33. Символ 9
D10809	WORD	Память для хранения названий рецептов. Задание 33. Символ 10
D10810	WORD	Память для хранения названий рецептов. Задание 33. Символ 11
D10811	WORD	Память для хранения названий рецептов. Задание 33. Символ 12
D10812	WORD	Память для хранения названий рецептов. Задание 33. Символ 13
D10813	WORD	Память для хранения названий рецептов. Задание 33. Символ 14
D10814	WORD	Память для хранения названий рецептов. Задание 33. Символ 15
D10815	WORD	Память для хранения названий рецептов. Задание 33. Символ 16
D10816	WORD	Память для хранения названий рецептов. Задание 33. Символ 17
D10817	WORD	Память для хранения названий рецептов. Задание 33. Символ 18
D10818	WORD	Память для хранения названий рецептов. Задание 33. Символ 19
D10819	WORD	Память для хранения названий рецептов. Задание 33. Символ 20
D10820	WORD	Память для хранения названий рецептов. Задание 33. Символ 21
D10821	WORD	Память для хранения названий рецептов. Задание 33. Символ 22
D10822	WORD	Память для хранения названий рецептов. Задание 33. Символ 23
D10823	WORD	Память для хранения названий рецептов. Задание 33. Символ 24
D10824	WORD	Память для хранения названий рецептов. Задание 33. Символ 25
D10825	WORD	Память для хранения названий рецептов. Задание 34. Символ 1
D10826	WORD	Память для хранения названий рецептов. Задание 34. Символ 2
D10827	WORD	Память для хранения названий рецептов. Задание 34. Символ 3
D10828	WORD	Память для хранения названий рецептов. Задание 34. Символ 4
D10829	WORD	Память для хранения названий рецептов. Задание 34. Символ 5
D10830	WORD	Память для хранения названий рецептов. Задание 34. Символ 6
D10831	WORD	Память для хранения названий рецептов. Задание 34. Символ 7
D10832	WORD	Память для хранения названий рецептов. Задание 34. Символ 8
D10833	WORD	Память для хранения названий рецептов. Задание 34. Символ 9
D10834	WORD	Память для хранения названий рецептов. Задание 34. Символ 10
D10835	WORD	Память для хранения названий рецептов. Задание 34. Символ 11
D10836	WORD	Память для хранения названий рецептов. Задание 34. Символ 12
D10837	WORD	Память для хранения названий рецептов. Задание 34. Символ 13
D10838	WORD	Память для хранения названий рецептов. Задание 34. Символ 14
D10839	WORD	Память для хранения названий рецептов. Задание 34. Символ 15
D10840	WORD	Память для хранения названий рецептов. Задание 34. Символ 16
D10841	WORD	Память для хранения названий рецептов. Задание 34. Символ 17
D10842	WORD	Память для хранения названий рецептов. Задание 34. Символ 18
D10843	WORD	Память для хранения названий рецептов. Задание 34. Символ 19
D10844	WORD	Память для хранения названий рецептов. Задание 34. Символ 20
D10845	WORD	Память для хранения названий рецептов. Задание 34. Символ 21
D10846	WORD	Память для хранения названий рецептов. Задание 34. Символ 22
D10847	WORD	Память для хранения названий рецептов. Задание 34. Символ 23
D10848	WORD	Память для хранения названий рецептов. Задание 34. Символ 24
D10849	WORD	Память для хранения названий рецептов. Задание 34. Символ 25
D10850	WORD	Память для хранения названий рецептов. Задание 35. Символ 1
D10851	WORD	Память для хранения названий рецептов. Задание 35. Символ 2
D10852	WORD	Память для хранения названий рецептов. Задание 35. Символ 3
D10853	WORD	Память для хранения названий рецептов. Задание 35. Символ 4
D10854	WORD	Память для хранения названий рецептов. Задание 35. Символ 5
D10855	WORD	Память для хранения названий рецептов. Задание 35. Символ 6
D10856	WORD	Память для хранения названий рецептов. Задание 35. Символ 7
D10857	WORD	Память для хранения названий рецептов. Задание 35. Символ 8
D10858	WORD	Память для хранения названий рецептов. Задание 35. Символ 9
D10859	WORD	Память для хранения названий рецептов. Задание 35. Символ 10
D10860	WORD	Память для хранения названий рецептов. Задание 35. Символ 11
D10861	WORD	Память для хранения названий рецептов. Задание 35. Символ 12
D10862	WORD	Память для хранения названий рецептов. Задание 35. Символ 13
D10863	WORD	Память для хранения названий рецептов. Задание 35. Символ 14
D10864	WORD	Память для хранения названий рецептов. Задание 35. Символ 15
D10865	WORD	Память для хранения названий рецептов. Задание 35. Символ 16
D10866	WORD	Память для хранения названий рецептов. Задание 35. Символ 17
D10867	WORD	Память для хранения названий рецептов. Задание 35. Символ 18
D10868	WORD	Память для хранения названий рецептов. Задание 35. Символ 19
D10869	WORD	Память для хранения названий рецептов. Задание 35. Символ 20
D10870	WORD	Память для хранения названий рецептов. Задание 35. Символ 21
D10871	WORD	Память для хранения названий рецептов. Задание 35. Символ 22
D10872	WORD	Память для хранения названий рецептов. Задание 35. Символ 23
D10873	WORD	Память для хранения названий рецептов. Задание 35. Символ 24
D10874	WORD	Память для хранения названий рецептов. Задание 35. Символ 25
D10875	WORD	Память для хранения названий рецептов. Задание 36. Символ 1
D10876	WORD	Память для хранения названий рецептов. Задание 36. Символ 2
D10877	WORD	Память для хранения названий рецептов. Задание 36. Символ 3
D10878	WORD	Память для хранения названий рецептов. Задание 36. Символ 4
D10879	WORD	Память для хранения названий рецептов. Задание 36. Символ 5
D10880	WORD	Память для хранения названий рецептов. Задание 36. Символ 6
D10881	WORD	Память для хранения названий рецептов. Задание 36. Символ 7
D10882	WORD	Память для хранения названий рецептов. Задание 36. Символ 8
D10883	WORD	Память для хранения названий рецептов. Задание 36. Символ 9
D10884	WORD	Память для хранения названий рецептов. Задание 36. Символ 10
D10885	WORD	Память для хранения названий рецептов. Задание 36. Символ 11
D10886	WORD	Память для хранения названий рецептов. Задание 36. Символ 12
D10887	WORD	Память для хранения названий рецептов. Задание 36. Символ 13
D10888	WORD	Память для хранения названий рецептов. Задание 36. Символ 14
D10889	WORD	Память для хранения названий рецептов. Задание 36. Символ 15
D10890	WORD	Память для хранения названий рецептов. Задание 36. Символ 16
D10891	WORD	Память для хранения названий рецептов. Задание 36. Символ 17
D10892	WORD	Память для хранения названий рецептов. Задание 36. Символ 18
D10893	WORD	Память для хранения названий рецептов. Задание 36. Символ 19
D10894	WORD	Память для хранения названий рецептов. Задание 36. Символ 20
D10895	WORD	Память для хранения названий рецептов. Задание 36. Символ 21
D10896	WORD	Память для хранения названий рецептов. Задание 36. Символ 22
D10897	WORD	Память для хранения названий рецептов. Задание 36. Символ 23
D10898	WORD	Память для хранения названий рецептов. Задание 36. Символ 24
D10899	WORD	Память для хранения названий рецептов. Задание 36. Символ 25
D10900	WORD	Память для хранения названий рецептов. Задание 37. Символ 1
D10901	WORD	Память для хранения названий рецептов. Задание 37. Символ 2
D10902	WORD	Память для хранения названий рецептов. Задание 37. Символ 3
D10903	WORD	Память для хранения названий рецептов. Задание 37. Символ 4
D10904	WORD	Память для хранения названий рецептов. Задание 37. Символ 5
D10905	WORD	Память для хранения названий рецептов. Задание 37. Символ 6
D10906	WORD	Память для хранения названий рецептов. Задание 37. Символ 7
D10907	WORD	Память для хранения названий рецептов. Задание 37. Символ 8
D10908	WORD	Память для хранения названий рецептов. Задание 37. Символ 9
D10909	WORD	Память для хранения названий рецептов. Задание 37. Символ 10
D10910	WORD	Память для хранения названий рецептов. Задание 37. Символ 11
D10911	WORD	Память для хранения названий рецептов. Задание 37. Символ 12
D10912	WORD	Память для хранения названий рецептов. Задание 37. Символ 13
D10913	WORD	Память для хранения названий рецептов. Задание 37. Символ 14
D10914	WORD	Память для хранения названий рецептов. Задание 37. Символ 15
D10915	WORD	Память для хранения названий рецептов. Задание 37. Символ 16
D10916	WORD	Память для хранения названий рецептов. Задание 37. Символ 17
D10917	WORD	Память для хранения названий рецептов. Задание 37. Символ 18
D10918	WORD	Память для хранения названий рецептов. Задание 37. Символ 19
D10919	WORD	Память для хранения названий рецептов. Задание 37. Символ 20
D10920	WORD	Память для хранения названий рецептов. Задание 37. Символ 21
D10921	WORD	Память для хранения названий рецептов. Задание 37. Символ 22
D10922	WORD	Память для хранения названий рецептов. Задание 37. Символ 23
D10923	WORD	Память для хранения названий рецептов. Задание 37. Символ 24
D10924	WORD	Память для хранения названий рецептов. Задание 37. Символ 25
D10925	WORD	Память для хранения названий рецептов. Задание 38. Символ 1
D10926	WORD	Память для хранения названий рецептов. Задание 38. Символ 2
D10927	WORD	Память для хранения названий рецептов. Задание 38. Символ 3
D10928	WORD	Память для хранения названий рецептов. Задание 38. Символ 4
D10929	WORD	Память для хранения названий рецептов. Задание 38. Символ 5
D10930	WORD	Память для хранения названий рецептов. Задание 38. Символ 6
D10931	WORD	Память для хранения названий рецептов. Задание 38. Символ 7
D10932	WORD	Память для хранения названий рецептов. Задание 38. Символ 8
D10933	WORD	Память для хранения названий рецептов. Задание 38. Символ 9
D10934	WORD	Память для хранения названий рецептов. Задание 38. Символ 10
D10935	WORD	Память для хранения названий рецептов. Задание 38. Символ 11
D10936	WORD	Память для хранения названий рецептов. Задание 38. Символ 12
D10937	WORD	Память для хранения названий рецептов. Задание 38. Символ 13
D10938	WORD	Память для хранения названий рецептов. Задание 38. Символ 14
D10939	WORD	Память для хранения названий рецептов. Задание 38. Символ 15
D10940	WORD	Память для хранения названий рецептов. Задание 38. Символ 16
D10941	WORD	Память для хранения названий рецептов. Задание 38. Символ 17
D10942	WORD	Память для хранения названий рецептов. Задание 38. Символ 18
D10943	WORD	Память для хранения названий рецептов. Задание 38. Символ 19
D10944	WORD	Память для хранения названий рецептов. Задание 38. Символ 20
D10945	WORD	Память для хранения названий рецептов. Задание 38. Символ 21
D10946	WORD	Память для хранения названий рецептов. Задание 38. Символ 22
D10947	WORD	Память для хранения названий рецептов. Задание 38. Символ 23
D10948	WORD	Память для хранения названий рецептов. Задание 38. Символ 24
D10949	WORD	Память для хранения названий рецептов. Задание 38. Символ 25
D10950	WORD	Память для хранения названий рецептов. Задание 39. Символ 1
D10951	WORD	Память для хранения названий рецептов. Задание 39. Символ 2
D10952	WORD	Память для хранения названий рецептов. Задание 39. Символ 3
D10953	WORD	Память для хранения названий рецептов. Задание 39. Символ 4
D10954	WORD	Память для хранения названий рецептов. Задание 39. Символ 5
D10955	WORD	Память для хранения названий рецептов. Задание 39. Символ 6
D10956	WORD	Память для хранения названий рецептов. Задание 39. Символ 7
D10957	WORD	Память для хранения названий рецептов. Задание 39. Символ 8
D10958	WORD	Память для хранения названий рецептов. Задание 39. Символ 9
D10959	WORD	Память для хранения названий рецептов. Задание 39. Символ 10
D11000	WORD	Память для хранения названий рецептов. Задание 41. Символ 1
D11001	WORD	Память для хранения названий рецептов. Задание 41. Символ 2
D11002	WORD	Память для хранения названий рецептов. Задание 41. Символ 3
D11003	WORD	Память для хранения названий рецептов. Задание 41. Символ 4
D11004	WORD	Память для хранения названий рецептов. Задание 41. Символ 5
D11005	WORD	Память для хранения названий рецептов. Задание 41. Символ 6
D11006	WORD	Память для хранения названий рецептов. Задание 41. Символ 7
D11007	WORD	Память для хранения названий рецептов. Задание 41. Символ 8
D11008	WORD	Память для хранения названий рецептов. Задание 41. Символ 9
D11009	WORD	Память для хранения названий рецептов. Задание 41. Символ 10
D11010	WORD	Память для хранения названий рецептов. Задание 41. Символ 11
D11011	WORD	Память для хранения названий рецептов. Задание 41. Символ 12
D11012	WORD	Память для хранения названий рецептов. Задание 41. Символ 13
D11013	WORD	Память для хранения названий рецептов. Задание 41. Символ 14
D11014	WORD	Память для хранения названий рецептов. Задание 41. Символ 15
D11015	WORD	Память для хранения названий рецептов. Задание 41. Символ 16
D11016	WORD	Память для хранения названий рецептов. Задание 41. Символ 17
